// TIA Portal project "项目1" (V14)

(* hardware
DEVICE "S7-1200 station_1"  S7-1200 Station
   slot 0: "Rack_0"  S7-1200 Rack  Rack  V1.0
   slot 1: "PLC_xingneng"  CPU 1214C DC/DC/DC  6ES7 214-1AG40-0XB0  V4.2
   slot 2: "DI 16/DQ 16x24VDC_1"  6ES7 223-1BL32-0XB0  V2.0
   slot 3: "DI 16/DQ 16x24VDC_2"  6ES7 223-1BL32-0XB0  V2.0
   slot 4: "AI 4x13BIT/AQ 2x14BIT_1"  6ES7 234-4HE32-0XB0  V2.0
   slot 5: "AI 4x13BIT/AQ 2x14BIT_2"  6ES7 234-4HE32-0XB0  V2.0
DEVICE "v90-pn-1"  GSD.Device.PN
   slot 0: "SINAMICS-V90-PN"  SINAMICS V90 PN V1.0  6SL3 210-5Fxxx-xxFx  V1.00
      slot 0: "SINAMICS V90 PN V1.0"  SINAMICS V90 PN V1.0
      slot 1: "驱动_1"  Drive
         slot 0: "模块访问点"  Module Access Point
         slot 1: "没有 PROFIsafe"  without PROFIsafe
      slot 1: "PN-IO"  PN-IO
         slot 1: "端口1"  Port 1
         slot 2: "端口2"  Port 2
   slot 0: "机架"  Rack  V1.0
   slot 2: "标准报文3, PZD-5/9"  Standard telegram 3, PZD-5/9
*)

// ===== PLC "PLC_xingneng"  CPU 1214C DC/DC/DC =====
// protected blocks, not shown: "buffer"

VAR_GLOBAL   // PLC tag table "默认变量表"
   "输入轴扭矩传感器" AT %IW128 : Int;
   "输出轴扭矩传感器Min_A" AT %IW130 : Int;
   "轴_1_LowHwLimitSwitch" AT %I0.3 : Bool;
   "轴_1_HighHwLimitSwitch" AT %I0.4 : Bool;
   "轴_1_参考点开关" AT %I0.2 : Bool;
   "轴_2_LowHwLimitSwitch" AT %I0.6 : Bool;
   "轴_2_HighHwLimitSwitch" AT %I0.7 : Bool;
   "轴_2_参考点开关" AT %I0.5 : Bool;
   "输出轴扭矩传感器Max_B" AT %IW132 : Int;
   "电流计" AT %IW134 : Int;
   "Tag_45" AT %I11.0 : Bool;
   "Tag_46" AT %I11.3 : Bool;
   "输入轴角度" AT %ID1000 : DInt;
   "Tag_70" AT %ID100 : DInt;
   "Tag_80" AT %ID0 : DWord;
   "Tag_86" AT %IW0 : Word;
   "Tag_87" AT %IW8 : Word;
   "Tag_88" AT %IW12 : Word;
   "工件在位" AT %I3.6 : Bool;
   "输入移报警" AT %I2.0 : Bool;
   "高度适配轴参考点" AT %I2.1 : Bool;
   "输出移报警" AT %I2.2 : Bool;
   "高度适配轴上限" AT %I2.3 : Bool;
   "输入旋报警" AT %I2.4 : Bool;
   "高度适配轴下限" AT %I2.5 : Bool;
   "输出旋报警" AT %I2.6 : Bool;
   "输出旋到位" AT %I2.7 : Bool;
   "抱花键进到位" AT %I3.0 : Bool;
   "抱花键退到位" AT %I3.1 : Bool;
   "摆臂1进到位" AT %I3.2 : Bool;
   "摆臂1退到位" AT %I3.3 : Bool;
   "摆臂2进到位" AT %I3.4 : Bool;
   "摆臂2退到位" AT %I3.5 : Bool;
   "振动进到位" AT %I4.0 : Bool;
   "振动退到位" AT %I4.1 : Bool;
   "升降门进到位" AT %I4.2 : Bool;
   "升降门退到位" AT %I4.3 : Bool;
   "急停" AT %I5.0 : Bool;
   "启动" AT %I5.1 : Bool;
   "复位" AT %I5.3 : Bool;
   "输出轴角度" AT %ID1004 : DInt;
   "Tag_1" AT %IW138 : Int;
   "ECU传感器" AT %IW136 : Int;
   "安全光栅" AT %I3.7 : Bool;
   "轴_5_Drive_IN" AT %I68.0 : "PD_TEL3_IN";
   "高度适配轴错误" AT %I1.5 : Bool;
   "产品定位缸进位" AT %I4.4 : Bool;
   "产品定位缸退位" AT %I4.5 : Bool;
   "右震动检测进位" AT %I4.6 : Bool;
   "右震动检测退位" AT %I4.7 : Bool;
   "Tag_116" AT %I5.4 : Bool;
   "工件在位检测" AT %I5.5 : Bool;
   "轴_1_Pulse_Up" AT %Q0.0 : Bool;
   "轴_1_Pulse_Down" AT %Q0.1 : Bool;
   "轴_2_脉冲" AT %Q0.2 : Bool;
   "轴_2_方向" AT %Q0.3 : Bool;
   "Tag_25" AT %QW128 : Word;
   "Tag_26" AT %QW130 : Int;
   "Tag_27" AT %QW80 : Int;
   "Tag_53" AT %Q6.0 : Bool;
   "Tag_54" AT %Q6.1 : Bool;
   "Tag_55" AT %Q6.2 : Bool;
   "Tag_56" AT %Q6.3 : Bool;
   "Tag_57" AT %Q6.4 : Bool;
   "Tag_58" AT %Q6.5 : Bool;
   "Tag_59" AT %Q6.6 : Bool;
   "Tag_60" AT %Q6.7 : Bool;
   "Tag_79" AT %QD0 : DWord;
   "Tag_82" AT %QW0 : Word;
   "Tag_83" AT %QW8 : Word;
   "Tag_84" AT %QW12 : Word;
   "Tag_85" AT %QW2 : Word;
   "控制器转速" AT %Q0.6 : Bool;
   "carPulse" AT %Q0.4 : Bool;
   "控制器切换" AT %Q1.0 : Bool;
   "输入移警清" AT %Q2.0 : Bool;
   "输出移警清" AT %Q2.1 : Bool;
   "输入旋模式" AT %Q2.3 : Bool;
   "输入旋警清" AT %Q2.4 : Bool;
   "输出旋模式" AT %Q2.6 : Bool;
   "输出旋警清" AT %Q2.7 : Bool;
   "抱花键" AT %Q4.0 : Bool;
   "摆臂进" AT %Q4.1 : Bool;
   "摆臂退" AT %Q4.2 : Bool;
   "振动" AT %Q4.5 : Bool;
   "升降门进" AT %Q4.3 : Bool;
   "升降门退" AT %Q4.4 : Bool;
   "黄" AT %Q3.0 : Bool;
   "绿" AT %Q3.1 : Bool;
   "红" AT %Q3.2 : Bool;
   "蜂鸣" AT %Q3.3 : Bool;
   "输入旋速" AT %Q2.2 : Bool;
   "输出旋速" AT %Q2.5 : Bool;
   "PowerECU" AT %Q0.5 : Bool;
   "switch" AT %Q3.5 : Bool;
   "0-1KHZ占空比" AT %QW132 : Int;
   "30V电源" AT %QW134 : Int;
   "Tag_7" AT %QD4 : DWord;
   "resetAxis1" AT %Q1.6 : Bool;
   "resetAxis2" AT %Q1.7 : Bool;
   "轴_4_方向" AT %Q0.7 : Bool;
   "轴_5_Drive_OUT" AT %Q64.0 : "PD_TEL3_OUT";
   "产品高度适配轴JOG+" AT %Q7.0 : Bool;
   "产品高度适配轴故障复位" AT %Q5.4 : Bool;
   "高度适配轴JOG+" AT %Q5.6 : Bool;
   "高度适配轴JOG-" AT %Q5.7 : Bool;
   "高度适配轴回原点" AT %Q5.5 : Bool;
   "产品定位缸进" AT %Q5.0 : Bool;
   "产品定位缸退" AT %Q5.1 : Bool;
   "右震动检测缸进" AT %Q5.2 : Bool;
   "右震动检测缸退" AT %Q5.3 : Bool;
   "电机方向" AT %Q4.6 : Bool;
   "电机控制" AT %Q4.7 : Bool;
   "funtionStatus" AT %MB10 : SInt;
   "Tag_18" AT %M0.0 : Bool;
   "Tag_19" AT %M0.1 : Bool;
   "Tag_20" AT %M0.2 : Bool;
   "Tag_21" AT %M0.3 : Bool;
   "Tag_22" AT %M0.7 : Bool;
   "Tag_23" AT %M0.6 : Bool;
   "Tag_24" AT %M0.4 : Bool;
   "Tag_30" AT %M0.5 : Bool;
   "torqueInput" AT %MD100 : Real;
   "torqueOutputA" AT %MD104 : Real;
   "Tag_33" AT %MD200 : Real;
   "Tag_34" AT %MD204 : Real;
   "Tag_35" AT %MD206 : Real;
   "Tag_36" AT %MD106 : Real;
   "torqueOutputB" AT %MD108 : Real;
   "current" AT %MD112 : Real;
   "Tag_3" AT %M10.0 : Bool;
   "Tag_42" AT %M11.0 : Bool;
   "Tag_43" AT %M12.0 : Bool;
   "Tag_44" AT %M10.1 : Bool;
   "Tag_47" AT %M10.2 : Bool;
   "Tag_48" AT %M10.3 : Bool;
   "Tag_51" AT %MW20 : Word;
   "Tag_62" AT %M10.4 : Bool;
   "Tag_64" AT %M10.5 : Bool;
   "Tag_65" AT %M12.3 : Bool;
   "Tag_66" AT %M13.0 : Bool;
   "Tag_67" AT %M11.1 : Bool;
   "Tag_68" AT %M10.6 : Bool;
   "Tag_69" AT %MW30 : Word;
   "Tag_71" AT %M30.0 : Bool;
   "Tag_72" AT %M35.0 : Bool;
   "Tag_73" AT %M30.5 : Bool;
   "Tag_74" AT %M35.6 : Bool;
   "Tag_75" AT %M35.5 : Bool;
   "Tag_76" AT %MW36 : Word;
   "Tag_77" AT %MW40 : Word;
   "Tag_89" AT %MW32 : Word;
   "Tag_28" AT %M30.7 : Bool;
   "Tag_29" AT %M1.0 : Bool;
   "Tag_49" AT %M1.1 : Bool;
   "Tag_50" AT %M1.2 : Bool;
   "Tag_61" AT %M1.3 : Bool;
   "Tag_90" AT %MB1 : Byte;
   "Tag_16" AT %M2.0 : Bool;
   "Tag_17" AT %M1.4 : Bool;
   "Tag_41" AT %M1.7 : Bool;
   "angleInput" AT %MD150 : Real;
   "angleOutput" AT %MD154 : Real;
   "sensorA" AT %MD116 : Real;
   "sensorB" AT %MD120 : Real;
   "carSpeed" AT %MD1000 : Real;
   "Tag_8" AT %M11.2 : Bool;
   "Tag_9" AT %M11.3 : Bool;
   "Tag_10" AT %M11.4 : Bool;
   "Tag_11" AT %M11.5 : Bool;
   "Tag_12" AT %M11.6 : Bool;
   "Tag_13" AT %M11.7 : Bool;
   "Tag_31" AT %M12.1 : Bool;
   "Tag_32" AT %M13.1 : Bool;
   "Tag_37" AT %M13.2 : Bool;
   "Tag_38" AT %M13.3 : Bool;
   "Tag_52" AT %M13.4 : Bool;
   "Tag_78" AT %M13.5 : Bool;
   "Tag_81" AT %M13.6 : Bool;
   "Tag_91" AT %M13.7 : Bool;
   "Tag_92" AT %MB11 : Byte;
   "Tag_93" AT %MB12 : Byte;
   "Tag_94" AT %MB13 : Byte;
   "Tag_95" AT %M2.1 : Bool;
   "carSpeed(1)" AT %MD5 : Real;
   "Tag_97" AT %M2.2 : Bool;
   "光栅故障" AT %M3.0 : Bool;
   "Tag_96" AT %M12.2 : Bool;
   "Tag_98" AT %MW1004 : Word;
   "Tag_99" AT %M300.0 : Bool;
   "Tag_100" AT %MW11 : Word;
   "Tag_101" AT %MD11 : DWord;
   "Tag_102" AT %M2.3 : Bool;
   "Tag_104" AT %M14.0 : Bool;
   "Tag_108" AT %M14.1 : Bool;
   "Tag_113" AT %M14.2 : Bool;
   "Tag_114" AT %M14.3 : Bool;
   "Tag_115" AT %M14.4 : Bool;
   "Tag_117" AT %M2.4 : Bool;
   "Tag_118" AT %M2.5 : Bool;
   "Tag_119" AT %M300.1 : Bool;
   "Tag_120" AT %M310.0 : Bool;
   "Tag_103" AT %M310.1 : Bool;
   "Tag_105" AT %M310.3 : Bool;
   "轴_5当前位移" AT %MD2000 : Real;
   "Tag_106" AT %M14.5 : Bool;
   "轴_1当前位移" AT %MD2004 : DWord;
   "轴_2当前位移" AT %MD2008 : DWord;
   "Tag_4" AT %M2012.0 : Bool;
   "Tag_5" AT %MD1004 : Real;
   "Tag_6" AT %MW2000 : Word;
   "Tag_107" AT %MW3000 : Word;
   "Tag_109" AT %MD2500 : DInt;
   "Tag_110" AT %MB2503 : Byte;
   "Tag_111" AT %M200.0 : Bool;
   "Tag_112" AT %M200.1 : Bool;
   "Tag_121" AT %M200.2 : Bool;
   "Tag_122" AT %M200.3 : Bool;
END_VAR

TYPE "In_config"
VERSION : 0.1
   STRUCT
      inAxis_接近位移 : Real;
      inAxis_接近速度 : Real;
      inAxis_套入位移 : Real;
      inAxis_套入速度 : Real;
      outAxis_接近位置 : Real;
      outAxis_接近速度 : Real;
      outAxis_套入位置 : Real;
      outAxis_套入速度 : Real;
   END_STRUCT;
END_TYPE

TYPE "In_swing_config"
VERSION : 0.1
   STRUCT
      启用状态 : Real;
      摆动速度 : Real;
      摆动角度 : Real;
      保护扭矩 : Real;
   END_STRUCT;
END_TYPE

TYPE "Fixture_transfer_config"
VERSION : 0.1
   STRUCT
      定位位置 : Real;
      定位速度 : Real;
   END_STRUCT;
END_TYPE

TYPE "Test_No_Load_CFG"
VERSION : 0.1
   STRUCT
      启用助力 : Real := 0.0;
      空载速度 : Real := 0.0;
      空载位移 : Real := 0.0;
      扭矩保护 : Real := 0.0;
   END_STRUCT;
END_TYPE

TYPE "Test_Function_CFG"
VERSION : 0.1
   STRUCT
      试验速度 : Real;
      试验角度 : Real;
      负载扭矩 : Real;
      保护扭矩 : Real;
   END_STRUCT;
END_TYPE

TYPE "Test_Input&Output_Characteristics_CFG"
VERSION : 0.1
   STRUCT
      试验速度 : Real;
      换向扭矩 : Real;
      模拟车速 : Real;
      模拟转速 : Real;
   END_STRUCT;
END_TYPE

TYPE "Test_NVH"
VERSION : 0.1
   STRUCT
      检测点1 : Real;
      检测点2 : Real;
      正向检测时间 : Real;
      逆向检测时间 : Real;
   END_STRUCT;
END_TYPE

DATA_BLOCK "auto_4_DB_1"   // DB1
{ S7_Optimized_Access := 'TRUE' }
VERSION : 0.1
// stored: InstanceOfName 逆向空载
"逆向空载"
BEGIN
END_DATA_BLOCK

DATA_BLOCK "Data_sendset"   // DB2
{ S7_Optimized_Access := 'TRUE' }
VERSION : 0.1
   VAR
      REQ : Bool;
      CONT : Bool := 1;
      LEN : UInt := 8;
      DONE : Bool;
      BUSY : Bool;
      ERROR : Bool;
      STATUS : Word;
      COM_RST : Bool;
      CONNECT : TCON_Param;
      NUM : DInt;
      X : Real;
      Y : Real;
      Z : Real;
   END_VAR
BEGIN
END_DATA_BLOCK

DATA_BLOCK "Data_send_0"   // DB3
{ S7_Optimized_Access := 'FALSE' }
VERSION : 0.1
   VAR
      ai : Array[0..99] of Real;
   END_VAR
BEGIN
END_DATA_BLOCK

DATA_BLOCK "auto_6_DB"   // DB4
{ S7_Optimized_Access := 'TRUE' }
VERSION : 0.1
// stored: InstanceOfName 固定工件
"固定工件"
BEGIN
END_DATA_BLOCK

DATA_BLOCK "Data_send_1"   // DB5
{ S7_Optimized_Access := 'FALSE' }
VERSION : 0.1
   VAR
      ai : Array[0..99] of Real;
   END_VAR
BEGIN
END_DATA_BLOCK

DATA_BLOCK "reset_DB"   // DB6
{ S7_Optimized_Access := 'TRUE' }
VERSION : 0.1
// stored: InstanceOfName reset
"reset"
BEGIN
END_DATA_BLOCK

DATA_BLOCK "MD_data"   // DB7
{ S7_Optimized_Access := 'FALSE' }
VERSION : 0.1
   VAR
      输入扭矩传感器参数 : Array[0..1] of Real;
      输出扭矩传感器参数A : Array[0..1] of Real;
      输出扭矩传感器参数B : Array[0..1] of Real;
      电流传感器参数 : Array[0..1] of Real;
      轴自动参数 : "In_config";
      输入轴移栽手动速度 : Array[0..3] of Real;
      输入轴旋转参数 : Array[0..3] of Real;
      工装定位参数 : "Fixture_transfer_config";
      工装手动参数 : Array[0..3] of Real;
      空载试验参数 : "Test_No_Load_CFG";
      功能试验参数 : "Test_Function_CFG";
      力特性试验参数 : "Test_Input&Output_Characteristics_CFG";
      逆向空载试验参数 : "Test_No_Load_CFG";
      振动NVH试验参数 : "Test_NVH";
      辅助参数 : Array[0..3] of Real;
   END_VAR
BEGIN
   输入扭矩传感器参数[1] := 18.8;   // 校验值19.2
   输出扭矩传感器参数A[1] := 10.0;   // 校验值9.5
   输出扭矩传感器参数B[1] := 113.0;   // 校验值97.0
   电流传感器参数[0] := -100.0;
   电流传感器参数[1] := 100.0;
   // 辅助参数[0] : 安全门开启
END_DATA_BLOCK

DATA_BLOCK "Data_recset"   // DB8
{ S7_Optimized_Access := 'TRUE' }
VERSION : 0.1
   VAR
      REQ : Bool;
      CONT : Bool := 1;
      LEN : UInt := 8;
      DONE : Bool;
      BUSY : Bool;
      ERROR : Bool;
      STATUS : Word;
      COM_RST : Bool;
      CONNECT : TCON_Param;
      NUM : UDInt;
      X : Real;
      Y : Real;
      Z : Real;
   END_VAR
BEGIN
END_DATA_BLOCK

DATA_BLOCK "alarm_DB"   // DB10
{ S7_Optimized_Access := 'TRUE' }
VERSION : 0.1
// stored: InstanceOfName alarm
"alarm"
BEGIN
END_DATA_BLOCK

DATA_BLOCK "auto_7_DB"   // DB12
{ S7_Optimized_Access := 'TRUE' }
VERSION : 0.1
// stored: InstanceOfName 振动检测
"振动检测"
BEGIN
END_DATA_BLOCK

DATA_BLOCK "Data_set"   // DB21
{ S7_Optimized_Access := 'TRUE' }
VERSION : 0.1
   VAR
      "real" : Array[0..16] of Real;
   END_VAR
BEGIN
   "real"[0] := 2.0;
END_DATA_BLOCK

DATA_BLOCK "manual_DB"   // DB22
{ S7_Optimized_Access := 'TRUE' }
VERSION : 0.1
// stored: InstanceOfName manual
"manual"
BEGIN
END_DATA_BLOCK

DATA_BLOCK "auto_8_DB"   // DB23
{ S7_Optimized_Access := 'TRUE' }
VERSION : 0.1
// stored: InstanceOfName 功能
"功能"
BEGIN
END_DATA_BLOCK

DATA_BLOCK "auto_1_DB"   // DB28
{ S7_Optimized_Access := 'TRUE' }
VERSION : 0.1
// stored: InstanceOfName 套输入轴花键
"套输入轴花键"
BEGIN
END_DATA_BLOCK

DATA_BLOCK "auto_2_DB"   // DB31
{ S7_Optimized_Access := 'TRUE' }
VERSION : 0.1
// stored: InstanceOfName 套输出轴花键
"套输出轴花键"
BEGIN
END_DATA_BLOCK

DATA_BLOCK "motor_run_DB"   // DB32
{ S7_Optimized_Access := 'TRUE' }
VERSION : 0.1
// stored: InstanceOfName motor_m
"motor_m"
BEGIN
END_DATA_BLOCK

DATA_BLOCK "motor_run_DB_1"   // DB33
{ S7_Optimized_Access := 'TRUE' }
VERSION : 0.1
// stored: InstanceOfName motor_m
"motor_m"
BEGIN
END_DATA_BLOCK

DATA_BLOCK "motor_run_DB_2"   // DB34
{ S7_Optimized_Access := 'TRUE' }
VERSION : 0.1
// stored: InstanceOfName motor_m
"motor_m"
BEGIN
END_DATA_BLOCK

DATA_BLOCK "motor_m_DB"   // DB35
{ S7_Optimized_Access := 'TRUE' }
VERSION : 0.1
// stored: InstanceOfName motor_m
"motor_m"
BEGIN
END_DATA_BLOCK

DATA_BLOCK "auto_3_DB"   // DB37
{ S7_Optimized_Access := 'TRUE' }
VERSION : 0.1
// stored: InstanceOfName 空载与标定
"空载与标定"
BEGIN
END_DATA_BLOCK

DATA_BLOCK "auto_4_DB"   // DB39
{ S7_Optimized_Access := 'TRUE' }
VERSION : 0.1
// stored: InstanceOfName 力特性
"力特性"
BEGIN
END_DATA_BLOCK

DATA_BLOCK "auto_100_DB"   // DB45
{ S7_Optimized_Access := 'TRUE' }
VERSION : 0.1
// stored: InstanceOfName auto_100
"auto_100"
BEGIN
END_DATA_BLOCK

DATA_BLOCK "找零_DB"   // DB66
{ S7_Optimized_Access := 'TRUE' }
VERSION : 0.1
// stored: InstanceOfName 找零
"找零"
BEGIN
END_DATA_BLOCK

DATA_BLOCK "MD_data_Rapid"   // DB70
{ S7_Optimized_Access := 'FALSE' }
VERSION : 0.1
   VAR
      设备编号 : Int;
      产品型号 : Int;
      设备状态 : Int;
      错误代码 : Int;
      当前曲线 : Int;
      传感器标定值 : Array[0..11] of Real;
   END_VAR
BEGIN
   // 传感器标定值[0] : 输入轴驱动伺服位移
   // 传感器标定值[1] : 输入轴移载伺服位移
   // 传感器标定值[2] : 工装移载伺服位移
   // 传感器标定值[3] : 输入轴旋转角度
   // 传感器标定值[4] : 输入轴扭矩
   // 传感器标定值[5] : 输出轴扭矩小量程
   // 传感器标定值[6] : 输出轴扭矩大量程
   // 传感器标定值[7] : 吸收电流
   // 传感器标定值[8] : factorSensorT1
   // 传感器标定值[9] : 输出轴旋转角度
   // 传感器标定值[10] : 输出轴移栽位移
   // 传感器标定值[11] : factorSensorT2
END_DATA_BLOCK

DATA_BLOCK "buffer_dataSet"   // DB100
{ S7_Optimized_Access := 'FALSE' }
VERSION : 0.1
   VAR
      factorInputTorque : Real := 20.0;
      factorOutputTorqueA : Real := 10.0;
      factorOutputTorqueB : Real := 100.0;
      factorCurrent : Real := 100.0;
      factorSensor : Real := 20.0;
      offsetInputTorqueRight : Real;
      offsetInputTorqueLeft : Real;
      offsetOutputTorqueRightA : Real;
      offsetOutputTorqueLeftA : Real;
      offsetOutputTorqueRightB : Real;
      offsetOutputTorqueLeftB : Real;
      offsetCurrent : Real;
      offsetSensor : Real;
      set_7 : Real;
      set_8 : Real;
      set_9 : Real;
      set_10 : Real;
      set_11 : Real;
      set_12 : Real;
      set_13 : Real;
      distanceInputNear : Real;
      distanceOutputNear : Real;
      distanceInputPoint : Real;
      distanceOutputPoint : Real;
      door : Real;
      voltageECU : Real;
      funtionSpeed : Real;
      funtionAngle : Real;
      funtionSpeedCar : Real;
      funtionLoad : Real;
      forceTorque : Real;
      noloadSpeed : Real;
      noloadAngle : Real;
      noloadPowerECU : Real;
      reverseloadSpeed : Real;
      reverseloadAngle : Real;
      reverseloadPowerECU : Real;
   END_VAR
BEGIN
END_DATA_BLOCK

DATA_BLOCK "buffer_dataSend"   // DB101
{ S7_Optimized_Access := 'FALSE' }
VERSION : 0.1
   VAR
      dataSend : Array[0..51] of Real;
   END_VAR
BEGIN
END_DATA_BLOCK

// folder: System blocks/Program resources

DATA_BLOCK "IEC_Timer_0_DB_1"   // DB51
{ S7_Optimized_Access := 'TRUE' }
AUTHOR : Simatic
FAMILY : IEC
NAME : IEC_TMR
VERSION : 1.0
// stored: InstanceOfName IEC_TIMER
"IEC_TIMER"
BEGIN
END_DATA_BLOCK

DATA_BLOCK "IEC_Timer_0_DB_3"   // DB59
{ S7_Optimized_Access := 'TRUE' }
AUTHOR : Simatic
FAMILY : IEC
NAME : IEC_TMR
VERSION : 1.0
// stored: InstanceOfName IEC_TIMER
"IEC_TIMER"
BEGIN
END_DATA_BLOCK

DATA_BLOCK "IEC_Timer_0_DB_4"   // DB63
{ S7_Optimized_Access := 'TRUE' }
AUTHOR : Simatic
FAMILY : IEC
NAME : IEC_TMR
VERSION : 1.0
// stored: InstanceOfName IEC_TIMER
"IEC_TIMER"
BEGIN
END_DATA_BLOCK

DATA_BLOCK "IEC_Timer_0_DB_2"   // DB64
{ S7_Optimized_Access := 'TRUE' }
AUTHOR : Simatic
FAMILY : IEC
NAME : IEC_TMR
VERSION : 1.0
// stored: InstanceOfName IEC_TIMER
"IEC_TIMER"
BEGIN
END_DATA_BLOCK

DATA_BLOCK "IEC_Timer_0_DB_5"   // DB65
{ S7_Optimized_Access := 'TRUE' }
AUTHOR : Simatic
FAMILY : IEC
NAME : IEC_TMR
VERSION : 1.0
// stored: InstanceOfName IEC_TIMER
"IEC_TIMER"
BEGIN
END_DATA_BLOCK

// folder: (top level)

DATA_BLOCK "轴_1"   // DB14, Motion_DB
{ S7_Optimized_Access := 'TRUE' }
AUTHOR : SIMATIC
FAMILY : BasicMC
NAME : TO_PosAx
VERSION : 6.0
// stored: InstanceOfName TO_PositioningAxis
"TO_PositioningAxis"
BEGIN
   // Axis.DirectionOutputEnabledCU = TRUE
   // Axis.OnlinePtoModeCUEnumValue = PTO（脉冲 A 和方向 B）
   // Axis.OnlinePtoModeCU = 16#0000_0002
   // Axis.SelectPTO = 0
   // Axis.LeadScrew = 5.0
   // Axis.LeadScrew.Distance = 1013
   // Axis.PositionLimitsMinPosition = -10000.0
   // Axis.PositionLimitsMinPosition.Distance = 1013
   // Axis.PositionLimitsMaxPosition = 10000.0
   // Axis.PositionLimitsMaxPosition.Distance = 1013
   // Axis.HomingOffset = 0.0
   // Axis.HomingOffset.Distance = 1013
   // Axis.HomingFastVelocity = 30.0
   // Axis.HomingFastVelocity.Distance = 1013
   // Axis.NormalizedMaxVelocity = 50.0
   // Axis.NormalizedMaxVelocity.Distance = 1013
   // Axis.NormalizedMaxVelocity.Time = 0
   // Axis.MaxVelocityReadOnly = 50.0
   // Axis.MaxVelocityReadOnly.Distance = 1013
   // Axis.NormalizedMinVelocity = 1.0
   // Axis.NormalizedMinVelocity.Distance = 1013
   // Axis.NormalizedMinVelocity.Time = 0
   // Axis.MinVelocityReadOnly = 1.0
   // Axis.MinVelocityReadOnly.Distance = 1013
   // Axis.Acceleration = 245.0
   // Axis.Acceleration.Distance = 1013
   // Axis.RampUpTime = 0.2
   // Axis.Deceleration = 245.0
   // Axis.Deceleration.Distance = 1013
   // Axis.RampDownTime = 0.2
   // Axis.RoundUpTime = 0.0
   // Axis.Jerk = 0.0
   // Axis.Jerk.Distance = 1013
   // Axis.RampDownTimeEmergency = 0.1
   // Axis.DecelerationEmergency = 490.0
   // Axis.DecelerationEmergency.Distance = 1013
   // Axis.HomingSlowVelocity = 10.0
   // Axis.HomingSlowVelocity.Distance = 1013
   // Axis.LengthUnitNormalized.Distance = 1013
   // Axis.LengthUnitNormalized.Time = 0
   // Pulse.OutputSourceCU = 16#0000_0000
   // Pulse.MaxFrequencyCU = 100000.0
   // Pulse.MinFrequencyCU = 1.0
   // Pulse.MaxDeltaFrequencyCU = 9.5E+9
   // Pulse.MinDeltaFrequencyCU = 0.005
   // Pulse.MaxDeltaDeltaFrequencyCU = 1.0E+10
   // Pulse.MinDeltaDeltaFrequencyCU = 0.004
   // Axis.SelectedChannel1EnumCU = %Q0.0
   // Axis.SelectedChannel2EnumCU = %Q0.1
   // Axis.PositionLimitsMin_AddressCU = %I0.3
   // Axis.PositionLimitsMax_AddressCU = %I0.4
   // Axis.PassiveHomingReferencePointSwitch_AddressCU = %I0.2
   // Axis.HomingReferencePointSwitch_AddressCU = %I0.2
END_DATA_BLOCK

DATA_BLOCK "轴_2"   // DB15, Motion_DB
{ S7_Optimized_Access := 'TRUE' }
AUTHOR : SIMATIC
FAMILY : BasicMC
NAME : TO_PosAx
VERSION : 6.0
// stored: InstanceOfName TO_PositioningAxis
"TO_PositioningAxis"
BEGIN
   // Axis.DirectionOutputEnabledCU = TRUE
   // Axis.OnlinePtoModeCUEnumValue = PTO（脉冲 A 和方向 B）
   // Axis.OnlinePtoModeCU = 16#0000_0002
   // Axis.SelectPTO = 1
   // Axis.LeadScrew = 5.0
   // Axis.LeadScrew.Distance = 1013
   // Axis.PositionLimitsMinPosition = -10000.0
   // Axis.PositionLimitsMinPosition.Distance = 1013
   // Axis.PositionLimitsMaxPosition = 10000.0
   // Axis.PositionLimitsMaxPosition.Distance = 1013
   // Axis.HomingOffset = 0.0
   // Axis.HomingOffset.Distance = 1013
   // Axis.HomingFastVelocity = 20.0
   // Axis.HomingFastVelocity.Distance = 1013
   // Axis.NormalizedMaxVelocity = 50.0
   // Axis.NormalizedMaxVelocity.Distance = 1013
   // Axis.NormalizedMaxVelocity.Time = 0
   // Axis.MaxVelocityReadOnly = 50.0
   // Axis.MaxVelocityReadOnly.Distance = 1013
   // Axis.NormalizedMinVelocity = 1.0
   // Axis.NormalizedMinVelocity.Distance = 1013
   // Axis.NormalizedMinVelocity.Time = 0
   // Axis.MinVelocityReadOnly = 1.0
   // Axis.MinVelocityReadOnly.Distance = 1013
   // Axis.Acceleration = 245.0
   // Axis.Acceleration.Distance = 1013
   // Axis.RampUpTime = 0.2
   // Axis.Deceleration = 245.0
   // Axis.Deceleration.Distance = 1013
   // Axis.RampDownTime = 0.2
   // Axis.RoundUpTime = 0.0
   // Axis.Jerk = 0.0
   // Axis.Jerk.Distance = 1013
   // Axis.RampDownTimeEmergency = 0.1
   // Axis.DecelerationEmergency = 490.0
   // Axis.DecelerationEmergency.Distance = 1013
   // Axis.HomingSlowVelocity = 10.0
   // Axis.HomingSlowVelocity.Distance = 1013
   // Axis.LengthUnitNormalized.Distance = 1013
   // Axis.LengthUnitNormalized.Time = 0
   // Pulse.OutputSourceCU = 16#0000_0000
   // Pulse.MaxFrequencyCU = 100000.0
   // Pulse.MinFrequencyCU = 1.0
   // Pulse.MaxDeltaFrequencyCU = 9.5E+9
   // Pulse.MinDeltaFrequencyCU = 0.005
   // Pulse.MaxDeltaDeltaFrequencyCU = 1.0E+10
   // Pulse.MinDeltaDeltaFrequencyCU = 0.004
   // Axis.OnlinePtoIndexCU = 1
   // Axis.SelectedChannel1EnumCU = %Q0.2
   // Axis.SelectedChannel2EnumCU = %Q0.3
   // Axis.PositionLimitsMin_AddressCU = %I0.6
   // Axis.PositionLimitsMax_AddressCU = %I0.7
   // Axis.PassiveHomingReferencePointSwitch_AddressCU = %I0.5
   // Axis.HomingReferencePointSwitch_AddressCU = %I0.5
END_DATA_BLOCK

DATA_BLOCK "轴_3"   // DB46, Motion_DB
{ S7_Optimized_Access := 'TRUE' }
AUTHOR : SIMATIC
FAMILY : BasicMC
NAME : TO_PosAx
VERSION : 6.0
// stored: InstanceOfName TO_PositioningAxis
"TO_PositioningAxis"
BEGIN
   // Axis.SelectedChannel2EnumCU = %Q0.3
   // Axis.OnlinePtoModeCUEnumValue = PTO（脉冲 A 和方向 B）
   // Axis.OnlinePtoModeCU = 16#0000_0002
   // Axis.SelectPTO = 2
   // Axis.LengthUnit.LastDistance = -1
   // Axis.LeadScrew = 10.0
   // Axis.LeadScrew.Distance = -1
   // Axis.PositionLimitsMinPosition = -1.0E+6
   // Axis.PositionLimitsMinPosition.Distance = -1
   // Axis.PositionLimitsMaxPosition = 1.0E+6
   // Axis.PositionLimitsMaxPosition.Distance = -1
   // Axis.HomingOffset = 0.0
   // Axis.HomingOffset.Distance = -1
   // Axis.HomingFastVelocity = 20000.0
   // Axis.HomingFastVelocity.Distance = -1
   // Axis.NormalizedMaxVelocity = 500.0
   // Axis.NormalizedMaxVelocity.Distance = -1
   // Axis.NormalizedMaxVelocity.Time = 0
   // Axis.MaxVelocityReadOnly = 500.0
   // Axis.MaxVelocityReadOnly.Distance = -1
   // Axis.NormalizedMinVelocity = 1.0
   // Axis.NormalizedMinVelocity.Distance = -1
   // Axis.NormalizedMinVelocity.Time = 0
   // Axis.MinVelocityReadOnly = 1.0
   // Axis.MinVelocityReadOnly.Distance = -1
   // Axis.Acceleration = 4990.0
   // Axis.Acceleration.Distance = -1
   // Axis.RampUpTime = 0.1
   // Axis.Deceleration = 4990.0
   // Axis.Deceleration.Distance = -1
   // Axis.RampDownTime = 0.1
   // Axis.RoundUpTime = 0.0
   // Axis.Jerk = 0.0
   // Axis.Jerk.Distance = -1
   // Axis.RampDownTimeEmergency = 0.1
   // Axis.DecelerationEmergency = 4990.0
   // Axis.DecelerationEmergency.Distance = -1
   // Axis.HomingSlowVelocity = 4000.0
   // Axis.HomingSlowVelocity.Distance = -1
   // Axis.LengthUnitNormalized.Distance = -1
   // Axis.LengthUnitNormalized.Time = 0
   // Pulse.OutputSourceCU = 16#0000_0000
   // Pulse.MaxFrequencyCU = 30000.0
   // Pulse.MinFrequencyCU = 1.0
   // Pulse.MaxDeltaFrequencyCU = 9.5E+9
   // Pulse.MinDeltaFrequencyCU = 0.005
   // Pulse.MaxDeltaDeltaFrequencyCU = 1.0E+10
   // Pulse.MinDeltaDeltaFrequencyCU = 0.004
   // Axis.OnlinePtoIndexCU = 2
   // Axis.SelectedChannel1EnumCU = %Q0.4
END_DATA_BLOCK

DATA_BLOCK "轴_5"   // DB52, Motion_DB
{ S7_Optimized_Access := 'TRUE' }
AUTHOR : SIMATIC
FAMILY : BasicMC
NAME : TO_PosAx
VERSION : 6.0
// stored: InstanceOfName TO_PositioningAxis
"TO_PositioningAxis"
BEGIN
   // Axis.PositionLimitsMax_AddressCU = %I2.3
   // Axis.PositionLimitsMin_AddressCU = %I2.5
   // Axis.HomingReferencePointSwitch_AddressCU = %I2.1
   // Axis.Encoder.TelegramAddressOutCU = %Q64.0
   // Axis.Encoder.TelegramAddressInCU = %I68.0
   // Axis.Encoder.OutputAddress = 64
   // Axis.Encoder.InputAddress = 68
   // Axis.Encoder.DoNameCU = SINAMICS-V90-PN.驱动_1
   // Axis.Drive.OutputAddress = 64
   // Axis.Drive.InputAddress = 68
   // Axis.Drive.TelegramAddressOutCU = %Q64.0
   // Axis.Drive.TelegramAddressInCU = %I68.0
   // Axis.Drive.TelegramType = 2
   // Axis.Drive.DoNameCU = SINAMICS-V90-PN.驱动_1
   // Axis.LengthUnitNormalized.Distance = 1013
   // Axis.Encoder.SelectedHscIndexCU = -1
   // Axis.Encoder.DbTypeCU = Classic
   // Axis.Drive.DbTypeCU = Classic
END_DATA_BLOCK

DATA_BLOCK "轴_4"   // DB53, Motion_DB
{ S7_Optimized_Access := 'TRUE' }
AUTHOR : SIMATIC
FAMILY : BasicMC
NAME : TO_PosAx
VERSION : 6.0
// stored: InstanceOfName TO_PositioningAxis
"TO_PositioningAxis"
BEGIN
   // Axis.SelectedChannel2EnumCU = %Q0.7
   // Axis.LengthUnit.LastDistance = -1
   // Axis.OnlinePtoModeCUEnumValue = PTO（脉冲 A 和方向 B）
   // Axis.OnlinePtoModeCU = 16#0000_0002
   // Axis.SelectedChannel1EnumCU = %Q0.6
   // Pulse.MinDeltaDeltaFrequencyCU = 0.004
   // Pulse.MaxDeltaDeltaFrequencyCU = 1.0E+10
   // Pulse.MinDeltaFrequencyCU = 0.005
   // Pulse.MaxDeltaFrequencyCU = 9.5E+9
   // Pulse.MinFrequencyCU = 1.0
   // Pulse.MaxFrequencyCU = 30000.0
   // Pulse.OutputSourceCU = 16#0000_0000
   // Axis.SelectPTO = 3
   // Axis.OnlinePtoIndexCU = 3
END_DATA_BLOCK

FUNCTION_BLOCK "alarm"   // FB1, LAD
{ S7_Optimized_Access := 'TRUE' }
VERSION : 0.1
   VAR
      "tempI4.4" : Bool;
      "tempI4.5" : Bool;
      "time" : IEC_TIMER;
      time_1 : IEC_TIMER;
      time_2 : IEC_TIMER;
      time_3 : IEC_TIMER;
      time_4 : IEC_TIMER;
      time_5 : IEC_TIMER;
      time_6 : IEC_TIMER;
      time_7 : IEC_TIMER;
      time_8 : IEC_TIMER;
      time_9 : IEC_TIMER;
      IEC_Timer_0_Instance : TON_TIME;
      IEC_Timer_0_Instance_1 : TON_TIME;
   END_VAR
   VAR_TEMP   // added for the SCL form of the ladder/FBD networks
      _w1 : Bool;
      _w2 : Bool;
   END_VAR
BEGIN

REGION Network 1
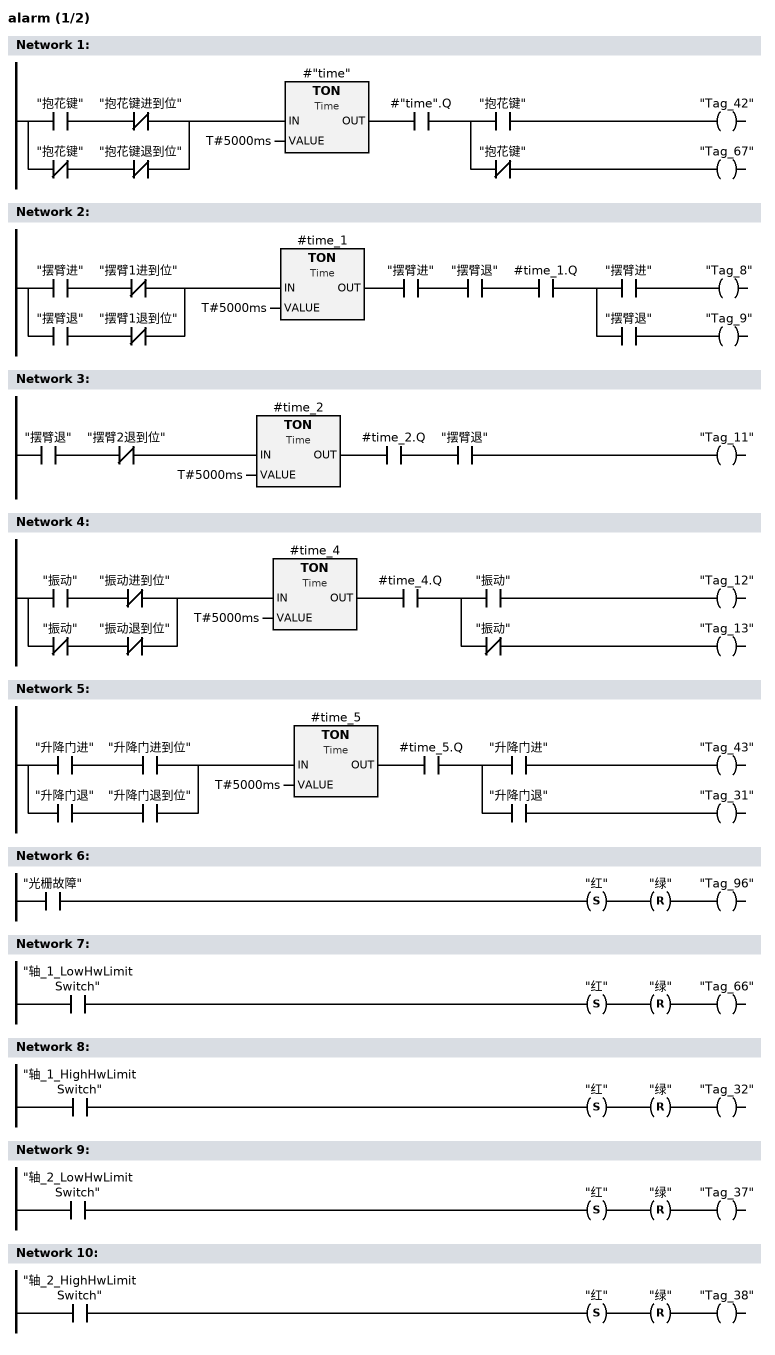
   #_w1 := ("抱花键" AND NOT "抱花键进到位") OR (NOT "抱花键" AND NOT "抱花键退到位");
   #"time".TON(IN := #_w1, PT := T#5000ms);   // TON coil
   #_w2 := #_w1 AND #"time".Q;
   "Tag_42" := #_w2 AND "抱花键";
   "Tag_67" := #_w2 AND NOT "抱花键";
END_REGION

REGION Network 2
   #_w1 := ("摆臂进" AND NOT "摆臂1进到位") OR ("摆臂退" AND NOT "摆臂1退到位");
   #time_1.TON(IN := #_w1, PT := T#5000ms);   // TON coil
   #_w2 := #_w1 AND "摆臂进" AND "摆臂退" AND #time_1.Q;
   "Tag_8" := #_w2 AND "摆臂进";
   "Tag_9" := #_w2 AND "摆臂退";
END_REGION

REGION Network 3
   #_w1 := "摆臂退" AND NOT "摆臂2退到位";
   #time_2.TON(IN := #_w1, PT := T#5000ms);   // TON coil
   "Tag_11" := #_w1 AND #time_2.Q AND "摆臂退";
END_REGION

REGION Network 4
   #_w1 := ("振动" AND NOT "振动进到位") OR (NOT "振动" AND NOT "振动退到位");
   #time_4.TON(IN := #_w1, PT := T#5000ms);   // TON coil
   #_w2 := #_w1 AND #time_4.Q;
   "Tag_12" := #_w2 AND "振动";
   "Tag_13" := #_w2 AND NOT "振动";
END_REGION

REGION Network 5
   #_w1 := ("升降门进" AND "升降门进到位") OR ("升降门退" AND "升降门退到位");
   #time_5.TON(IN := #_w1, PT := T#5000ms);   // TON coil
   #_w2 := #_w1 AND #time_5.Q;
   "Tag_43" := #_w2 AND "升降门进";
   "Tag_31" := #_w2 AND "升降门退";
END_REGION

REGION Network 6
   RUNG wire#powerrail
      Contact( "光栅故障" )
      S_Coil( "红" )
      R_Coil( "绿" )
      Coil( "Tag_96" )
   END_RUNG
   // the same network as SCL:
   IF "光栅故障" THEN
       "红" := TRUE;
       "绿" := FALSE;
   END_IF;
   "Tag_96" := "光栅故障";
END_REGION

REGION Network 7
   RUNG wire#powerrail
      Contact( "轴_1_LowHwLimitSwitch" )
      S_Coil( "红" )
      R_Coil( "绿" )
      Coil( "Tag_66" )
   END_RUNG
   // the same network as SCL:
   IF "轴_1_LowHwLimitSwitch" THEN
       "红" := TRUE;
       "绿" := FALSE;
   END_IF;
   "Tag_66" := "轴_1_LowHwLimitSwitch";
END_REGION

REGION Network 8
   RUNG wire#powerrail
      Contact( "轴_1_HighHwLimitSwitch" )
      S_Coil( "红" )
      R_Coil( "绿" )
      Coil( "Tag_32" )
   END_RUNG
   // the same network as SCL:
   IF "轴_1_HighHwLimitSwitch" THEN
       "红" := TRUE;
       "绿" := FALSE;
   END_IF;
   "Tag_32" := "轴_1_HighHwLimitSwitch";
END_REGION

REGION Network 9
   RUNG wire#powerrail
      Contact( "轴_2_LowHwLimitSwitch" )
      S_Coil( "红" )
      R_Coil( "绿" )
      Coil( "Tag_37" )
   END_RUNG
   // the same network as SCL:
   IF "轴_2_LowHwLimitSwitch" THEN
       "红" := TRUE;
       "绿" := FALSE;
   END_IF;
   "Tag_37" := "轴_2_LowHwLimitSwitch";
END_REGION

REGION Network 10
   RUNG wire#powerrail
      Contact( "轴_2_HighHwLimitSwitch" )
      S_Coil( "红" )
      R_Coil( "绿" )
      Coil( "Tag_38" )
   END_RUNG
   // the same network as SCL:
   IF "轴_2_HighHwLimitSwitch" THEN
       "红" := TRUE;
       "绿" := FALSE;
   END_IF;
   "Tag_38" := "轴_2_HighHwLimitSwitch";
END_REGION

REGION Network 12
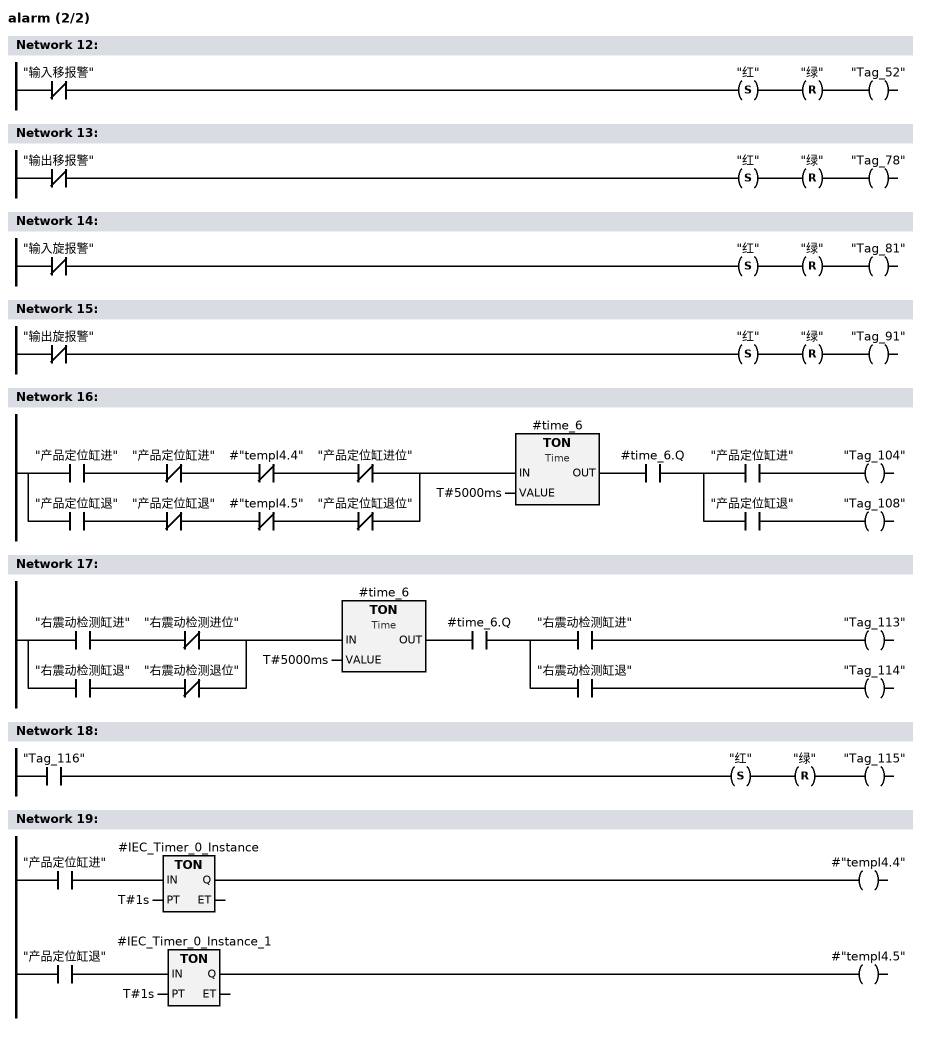
   RUNG wire#powerrail
      I_Contact( "输入移报警" )
      S_Coil( "红" )
      R_Coil( "绿" )
      Coil( "Tag_52" )
   END_RUNG
   // the same network as SCL:
   IF NOT "输入移报警" THEN
       "红" := TRUE;
       "绿" := FALSE;
   END_IF;
   "Tag_52" := NOT "输入移报警";
END_REGION

REGION Network 13
   RUNG wire#powerrail
      I_Contact( "输出移报警" )
      S_Coil( "红" )
      R_Coil( "绿" )
      Coil( "Tag_78" )
   END_RUNG
   // the same network as SCL:
   IF NOT "输出移报警" THEN
       "红" := TRUE;
       "绿" := FALSE;
   END_IF;
   "Tag_78" := NOT "输出移报警";
END_REGION

REGION Network 14
   RUNG wire#powerrail
      I_Contact( "输入旋报警" )
      S_Coil( "红" )
      R_Coil( "绿" )
      Coil( "Tag_81" )
   END_RUNG
   // the same network as SCL:
   IF NOT "输入旋报警" THEN
       "红" := TRUE;
       "绿" := FALSE;
   END_IF;
   "Tag_81" := NOT "输入旋报警";
END_REGION

REGION Network 15
   RUNG wire#powerrail
      I_Contact( "输出旋报警" )
      S_Coil( "红" )
      R_Coil( "绿" )
      Coil( "Tag_91" )
   END_RUNG
   // the same network as SCL:
   IF NOT "输出旋报警" THEN
       "红" := TRUE;
       "绿" := FALSE;
   END_IF;
   "Tag_91" := NOT "输出旋报警";
END_REGION

REGION Network 16
   #_w1 := ("产品定位缸进" AND NOT "产品定位缸进" AND NOT #"tempI4.4" AND NOT "产品定位缸进位") OR ("产品定位缸退" AND NOT "产品定位缸退" AND NOT #"tempI4.5" AND NOT "产品定位缸退位");
   #time_6.TON(IN := #_w1, PT := T#5000ms);   // TON coil
   #_w2 := #_w1 AND #time_6.Q;
   "Tag_104" := #_w2 AND "产品定位缸进";
   "Tag_108" := #_w2 AND "产品定位缸退";
END_REGION

REGION Network 17
   #_w1 := ("右震动检测缸进" AND NOT "右震动检测进位") OR ("右震动检测缸退" AND NOT "右震动检测退位");
   #time_6.TON(IN := #_w1, PT := T#5000ms);   // TON coil
   #_w2 := #_w1 AND #time_6.Q;
   "Tag_113" := #_w2 AND "右震动检测缸进";
   "Tag_114" := #_w2 AND "右震动检测缸退";
END_REGION

REGION Network 18
   RUNG wire#powerrail
      Contact( "Tag_116" )
      S_Coil( "红" )
      R_Coil( "绿" )
      Coil( "Tag_115" )
   END_RUNG
   // the same network as SCL:
   IF "Tag_116" THEN
       "红" := TRUE;
       "绿" := FALSE;
   END_IF;
   "Tag_115" := "Tag_116";
END_REGION

REGION Network 19
   #IEC_Timer_0_Instance(IN := "产品定位缸进", PT := T#1s);   // TON
   #"tempI4.4" := #IEC_Timer_0_Instance.Q;
   #IEC_Timer_0_Instance_1(IN := "产品定位缸退", PT := T#1s);   // TON
   #"tempI4.5" := #IEC_Timer_0_Instance_1.Q;
END_REGION
END_FUNCTION_BLOCK

FUNCTION_BLOCK "reset"   // FB2, LAD
{ S7_Optimized_Access := 'TRUE' }
VERSION : 0.1
   VAR_INPUT
      stt : Bool;
      stp : Bool;
   END_VAR
   VAR_OUTPUT
      done : Bool;
      error : Bool;
      busy : Bool;
   END_VAR
   VAR
      p1 : Real;
      p2 : Real;
      "m" : Array[0..100] of Bool;
      Done_1 : Array[0..5] of Bool;
      "time" : IEC_TIMER;
      IEC_Timer_0_Instance : TON_TIME;
      MC_Reset_Instance : MC_Reset;
      MC_Home_Instance : MC_Home;
      MC_MoveAbsolute_Instance : MC_MoveAbsolute;
      CTRL_HSC_0_Instance : CTRL_HSC;
   END_VAR
   VAR_TEMP
      done1 : Bool;
      done2 : Bool;
      done3 : Bool;
      done4 : Bool;
   END_VAR
   VAR_TEMP   // added for the SCL form of the ladder/FBD networks
      _w1 : Bool;
   END_VAR
BEGIN

REGION Network 1
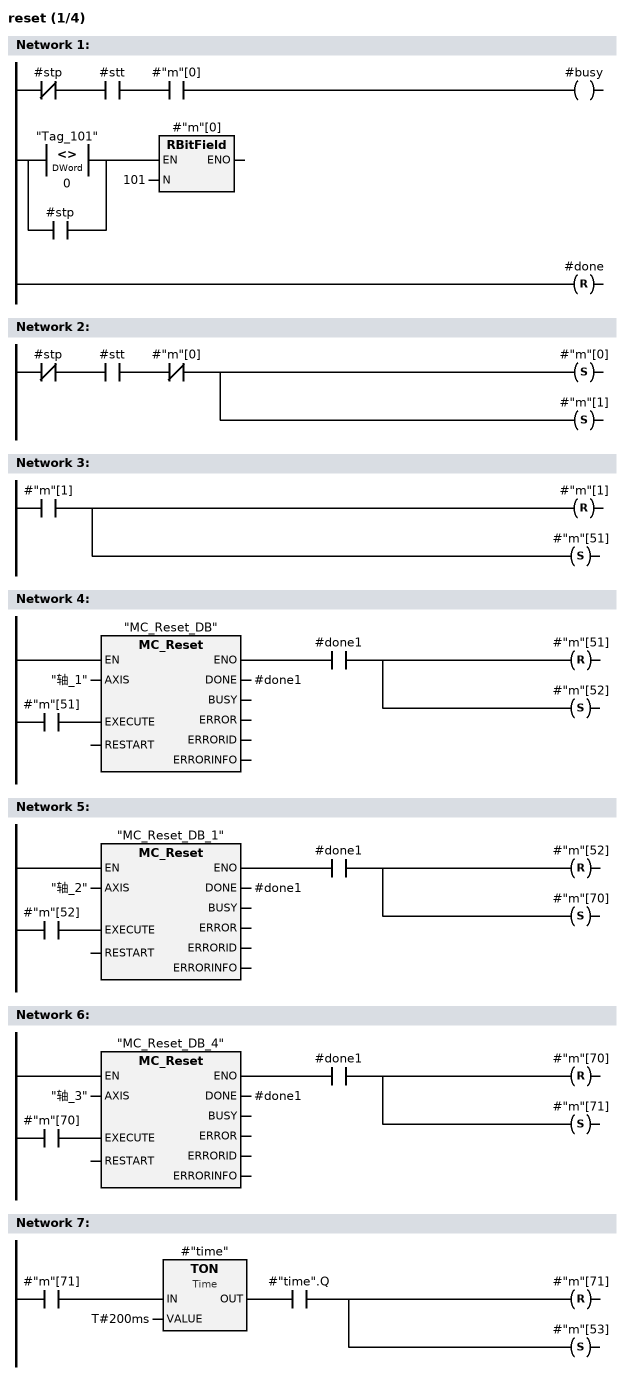
   // no SCL statement known for RBitField: written as a call
   #busy := NOT #stp AND #stt AND #"m"[0];
   IF ("Tag_101" <> 0) OR #stp THEN RBitField(n := 101, operand := #"m"[0]); END_IF;
   #done := FALSE;
END_REGION

REGION Network 2
   RUNG wire#powerrail
      I_Contact( #stp )
      Contact( #stt )
      I_Contact( #"m"[0] )
      wire#w1
      S_Coil( #"m"[0] )
   END_RUNG
   RUNG wire#w1
      S_Coil( #"m"[1] )
   END_RUNG
   // the same network as SCL:
   #_w1 := NOT #stp AND #stt AND NOT #"m"[0];
   IF #_w1 THEN
       #"m"[0] := TRUE;
       #"m"[1] := TRUE;
   END_IF;
END_REGION

REGION Network 3
   RUNG wire#powerrail
      Contact( #"m"[1] )
      wire#w1
      R_Coil( #"m"[1] )
   END_RUNG
   RUNG wire#w1
      S_Coil( #"m"[51] )
   END_RUNG
   // the same network as SCL:
   #_w1 := #"m"[1];
   IF #_w1 THEN
       #"m"[1] := FALSE;
       #"m"[51] := TRUE;
   END_IF;
END_REGION

REGION Network 4
   // ENO of a box is taken as its EN; it also drops when the box reports an error
   "MC_Reset_DB"(Axis := "轴_1", Execute := #"m"[51], Done => #done1);   // MC_Reset
   IF #done1 THEN
       #"m"[51] := FALSE;
       #"m"[52] := TRUE;
   END_IF;
END_REGION

REGION Network 5
   // ENO of a box is taken as its EN; it also drops when the box reports an error
   "MC_Reset_DB_1"(Axis := "轴_2", Execute := #"m"[52], Done => #done1);   // MC_Reset
   IF #done1 THEN
       #"m"[52] := FALSE;
       #"m"[70] := TRUE;
   END_IF;
END_REGION

REGION Network 6
   // ENO of a box is taken as its EN; it also drops when the box reports an error
   "MC_Reset_DB_4"(Axis := "轴_3", Execute := #"m"[70], Done => #done1);   // MC_Reset
   IF #done1 THEN
       #"m"[70] := FALSE;
       #"m"[71] := TRUE;
   END_IF;
END_REGION

REGION Network 7
   #"time".TON(IN := #"m"[71], PT := T#200ms);   // TON coil
   #_w1 := #"m"[71] AND #"time".Q;
   IF #_w1 THEN
       #"m"[71] := FALSE;
       #"m"[53] := TRUE;
   END_IF;
END_REGION

REGION Network 8
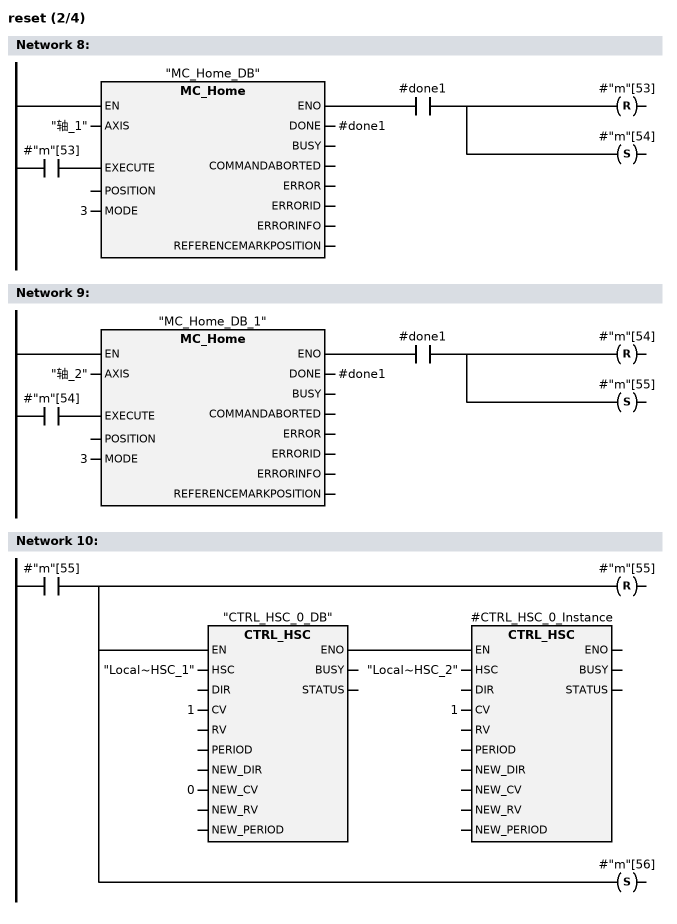
   // ENO of a box is taken as its EN; it also drops when the box reports an error
   "MC_Home_DB"(Axis := "轴_1", Execute := #"m"[53], Mode := 3, Done => #done1);   // MC_Home
   IF #done1 THEN
       #"m"[53] := FALSE;
       #"m"[54] := TRUE;
   END_IF;
END_REGION

REGION Network 9
   // ENO of a box is taken as its EN; it also drops when the box reports an error
   "MC_Home_DB_1"(Axis := "轴_2", Execute := #"m"[54], Mode := 3, Done => #done1);   // MC_Home
   IF #done1 THEN
       #"m"[54] := FALSE;
       #"m"[55] := TRUE;
   END_IF;
END_REGION

REGION Network 10
   // ENO of a box is taken as its EN; it also drops when the box reports an error
   #_w1 := #"m"[55];
   IF #_w1 THEN
       #"m"[55] := FALSE;
       "CTRL_HSC_0_DB"(HSC := "Local~HSC_1", CV := 1, NEW_CV := 0);   // CTRL_HSC
       #CTRL_HSC_0_Instance(HSC := "Local~HSC_2", CV := 1);   // CTRL_HSC
       #"m"[56] := TRUE;
   END_IF;
END_REGION

REGION Network 11
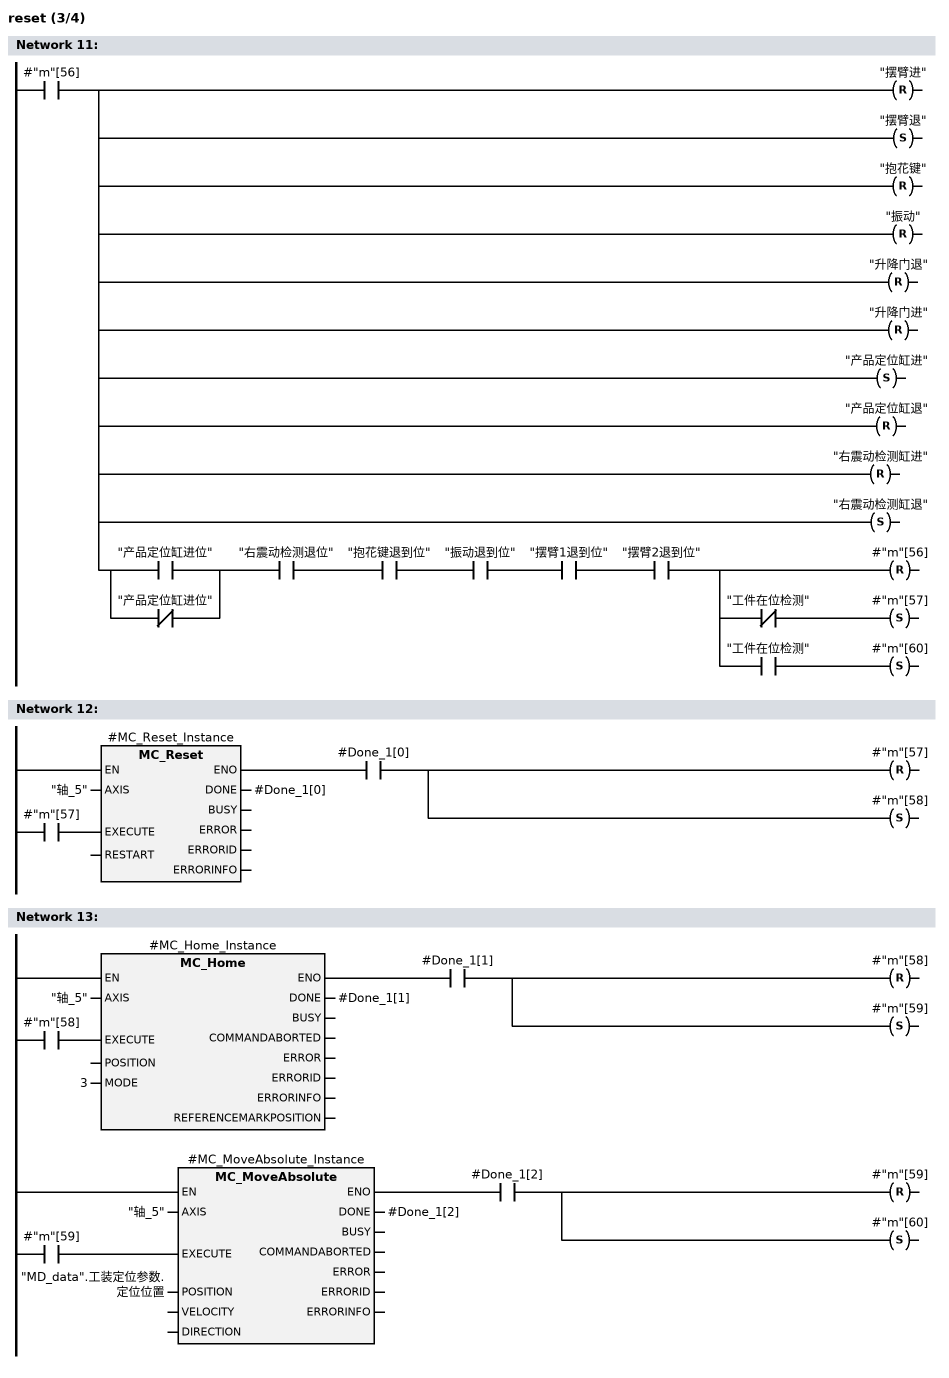
   RUNG wire#powerrail
      Contact( #"m"[56] )
      wire#w1
      R_Coil( "摆臂进" )
   END_RUNG
   RUNG wire#w1
      S_Coil( "摆臂退" )
   END_RUNG
   RUNG wire#w1
      R_Coil( "抱花键" )
   END_RUNG
   RUNG wire#w1
      R_Coil( "振动" )
   END_RUNG
   RUNG wire#w1
      R_Coil( "升降门退" )
   END_RUNG
   RUNG wire#w1
      R_Coil( "升降门进" )
   END_RUNG
   RUNG wire#w1
      S_Coil( "产品定位缸进" )
   END_RUNG
   RUNG wire#w1
      R_Coil( "产品定位缸退" )
   END_RUNG
   RUNG wire#w1
      R_Coil( "右震动检测缸进" )
   END_RUNG
   RUNG wire#w1
      S_Coil( "右震动检测缸退" )
   END_RUNG
   RUNG wire#w1
      Contact( "产品定位缸进位" )
      wire#w2
      Contact( "右震动检测退位" )
      Contact( "抱花键退到位" )
      Contact( "振动退到位" )
      Contact( "摆臂1退到位" )
      Contact( "摆臂2退到位" )
      wire#w3
      R_Coil( #"m"[56] )
   END_RUNG
   RUNG wire#w1
      I_Contact( "产品定位缸进位" )
   END_RUNG wire#w2
   RUNG wire#w3
      I_Contact( "工件在位检测" )
      S_Coil( #"m"[57] )
   END_RUNG
   RUNG wire#w3
      Contact( "工件在位检测" )
      S_Coil( #"m"[60] )
   END_RUNG
   // the same network as SCL:
   IF #"m"[56] THEN
       "摆臂进" := FALSE;
       "摆臂退" := TRUE;
       "抱花键" := FALSE;
       "振动" := FALSE;
       "升降门退" := FALSE;
       "升降门进" := FALSE;
       "产品定位缸进" := TRUE;
       "产品定位缸退" := FALSE;
       "右震动检测缸进" := FALSE;
       "右震动检测缸退" := TRUE;
   END_IF;
   #_w1 := #"m"[56] AND ("产品定位缸进位" OR NOT "产品定位缸进位") AND "右震动检测退位" AND "抱花键退到位" AND "振动退到位" AND "摆臂1退到位" AND "摆臂2退到位";
   IF #_w1 THEN #"m"[56] := FALSE; END_IF;
   IF #_w1 AND NOT "工件在位检测" THEN #"m"[57] := TRUE; END_IF;
   IF #_w1 AND "工件在位检测" THEN #"m"[60] := TRUE; END_IF;
END_REGION

REGION Network 12
   // ENO of a box is taken as its EN; it also drops when the box reports an error
   #MC_Reset_Instance(Axis := "轴_5", Execute := #"m"[57], Done => #Done_1[0]);   // MC_Reset
   IF #Done_1[0] THEN
       #"m"[57] := FALSE;
       #"m"[58] := TRUE;
   END_IF;
END_REGION

REGION Network 13
   // ENO of a box is taken as its EN; it also drops when the box reports an error
   #MC_Home_Instance(Axis := "轴_5", Execute := #"m"[58], Mode := 3, Done => #Done_1[1]);   // MC_Home
   IF #Done_1[1] THEN
       #"m"[58] := FALSE;
       #"m"[59] := TRUE;
   END_IF;
   #MC_MoveAbsolute_Instance(Axis := "轴_5",   // MC_MoveAbsolute
                           Execute := #"m"[59],
                           Position := "MD_data".工装定位参数.定位位置,
                           Done => #Done_1[2]);
   IF #Done_1[2] THEN
       #"m"[59] := FALSE;
       #"m"[60] := TRUE;
   END_IF;
END_REGION

REGION Network 14
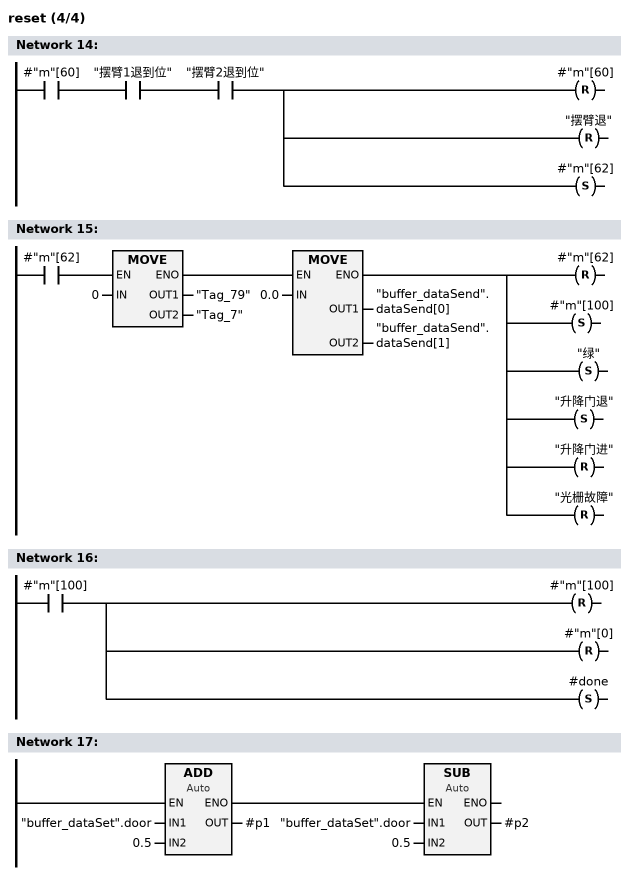
   RUNG wire#powerrail
      Contact( #"m"[60] )
      Contact( "摆臂1退到位" )
      Contact( "摆臂2退到位" )
      wire#w1
      R_Coil( #"m"[60] )
   END_RUNG
   RUNG wire#w1
      R_Coil( "摆臂退" )
   END_RUNG
   RUNG wire#w1
      S_Coil( #"m"[62] )
   END_RUNG
   // the same network as SCL:
   #_w1 := #"m"[60] AND "摆臂1退到位" AND "摆臂2退到位";
   IF #_w1 THEN
       #"m"[60] := FALSE;
       "摆臂退" := FALSE;
       #"m"[62] := TRUE;
   END_IF;
END_REGION

REGION Network 15
   RUNG wire#powerrail
      Contact( #"m"[62] )
      Move(in := 0, out1 => "Tag_79", out2 => "Tag_7")
      Move(in := 0.0, out1 => "buffer_dataSend".dataSend[0], out2 => "buffer_dataSend".dataSend[1])
      wire#w1
      R_Coil( #"m"[62] )
   END_RUNG
   RUNG wire#w1
      S_Coil( #"m"[100] )
   END_RUNG
   RUNG wire#w1
      S_Coil( "绿" )
   END_RUNG
   RUNG wire#w1
      S_Coil( "升降门退" )
   END_RUNG
   RUNG wire#w1
      R_Coil( "升降门进" )
   END_RUNG
   RUNG wire#w1
      R_Coil( "光栅故障" )
   END_RUNG
   // the same network as SCL:
   IF #"m"[62] THEN
       "Tag_79" := 0;
       "Tag_7" := 0;
       "buffer_dataSend".dataSend[0] := 0.0;
       "buffer_dataSend".dataSend[1] := 0.0;
   END_IF;
   #_w1 := #"m"[62];
   IF #_w1 THEN
       #"m"[62] := FALSE;
       #"m"[100] := TRUE;
       "绿" := TRUE;
       "升降门退" := TRUE;
       "升降门进" := FALSE;
       "光栅故障" := FALSE;
   END_IF;
END_REGION

REGION Network 16
   RUNG wire#powerrail
      Contact( #"m"[100] )
      wire#w1
      R_Coil( #"m"[100] )
   END_RUNG
   RUNG wire#w1
      R_Coil( #"m"[0] )
   END_RUNG
   RUNG wire#w1
      S_Coil( #done )
   END_RUNG
   // the same network as SCL:
   #_w1 := #"m"[100];
   IF #_w1 THEN
       #"m"[100] := FALSE;
       #"m"[0] := FALSE;
       #done := TRUE;
   END_IF;
END_REGION

REGION Network 17
   RUNG wire#powerrail
      Add(in1 := "buffer_dataSet".door, in2 := 0.5, out => #p1)
      Sub(in1 := "buffer_dataSet".door, in2 := 0.5, out => #p2)
   END_RUNG
   // the same network as SCL:
   #p1 := "buffer_dataSet".door + 0.5;
   #p2 := "buffer_dataSet".door - 0.5;
END_REGION
END_FUNCTION_BLOCK

FUNCTION_BLOCK "manual"   // FB3, LAD
{ S7_Optimized_Access := 'TRUE' }
VERSION : 0.1
   VAR_INPUT
      open : Bool;
      emg : Bool;
   END_VAR
   VAR
      temp_1 : Bool;
      temp_2 : Bool;
      buffer : Array[0..20] of Byte;
      emg_n : Bool;
      MC_MoveJog_Instance : MC_MoveJog;
      MC_Reset_Instance : MC_Reset;
      MC_Power_Instance : MC_Power;
      MC_Home_Instance : MC_Home;
      MC_MoveAbsolute_Instance : MC_MoveAbsolute;
      MC_Power_Instance_1 : MC_Power;
      IEC_Timer_0_Instance : TON_TIME;
      IEC_Timer_0_Instance_1 : TON_TIME;
      IEC_Timer_0_Instance_2 : TON_TIME;
      IEC_Timer_0_Instance_3 : TON_TIME;
      IEC_Timer_0_Instance_4 : TON_TIME;
      IEC_Timer_0_Instance_5 : TON_TIME;
      MC_Halt_Instance : MC_Halt;
   END_VAR
   VAR_TEMP
      "m" : Real;
      m_1 : Real;
   END_VAR
   VAR_TEMP   // added for the SCL form of the ladder/FBD networks
      _w1 : Bool;
      _w2 : Bool;
      _w3 : Bool;
      _w4 : Bool;
   END_VAR
BEGIN

REGION Network 2
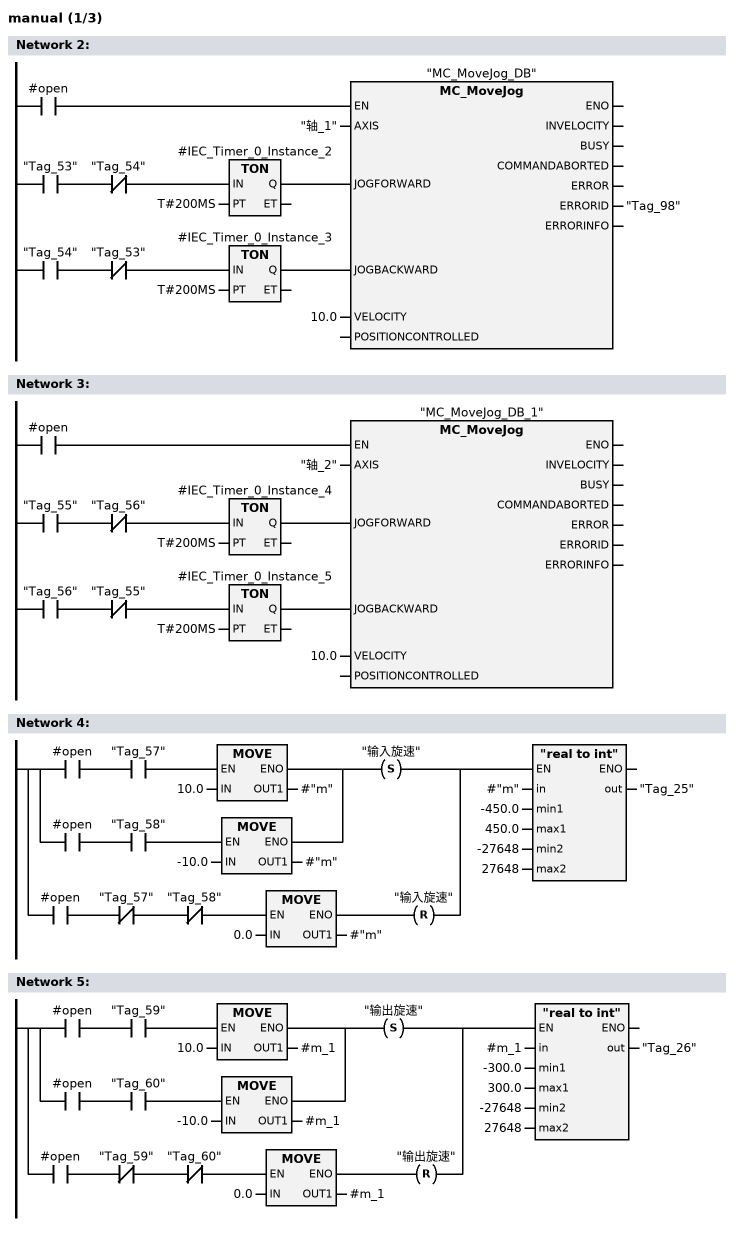
   #IEC_Timer_0_Instance_2(IN := "Tag_53" AND NOT "Tag_54", PT := T#200MS);   // TON
   #IEC_Timer_0_Instance_3(IN := "Tag_54" AND NOT "Tag_53", PT := T#200MS);   // TON
   IF #open THEN
       "MC_MoveJog_DB"(Axis := "轴_1",   // MC_MoveJog
                       JogForward := #IEC_Timer_0_Instance_2.Q,
                       JogBackward := #IEC_Timer_0_Instance_3.Q,
                       Velocity := 10.0,
                       ErrorID => "Tag_98");
   END_IF;
END_REGION

REGION Network 3
   #IEC_Timer_0_Instance_4(IN := "Tag_55" AND NOT "Tag_56", PT := T#200MS);   // TON
   #IEC_Timer_0_Instance_5(IN := "Tag_56" AND NOT "Tag_55", PT := T#200MS);   // TON
   IF #open THEN
       "MC_MoveJog_DB_1"(Axis := "轴_2",   // MC_MoveJog
                         JogForward := #IEC_Timer_0_Instance_4.Q,
                         JogBackward := #IEC_Timer_0_Instance_5.Q,
                         Velocity := 10.0);
   END_IF;
END_REGION

REGION Network 4
   RUNG wire#powerrail
      Contact( #open )
      Contact( "Tag_57" )
      Move(in := 10.0, out1 => #"m")
      wire#w1
      S_Coil( "输入旋速" )
      wire#w2
      "real to int"(in := #"m", min1 := -450.0, max1 := 450.0, min2 := -27648, max2 := 27648, out => "Tag_25")
   END_RUNG
   RUNG wire#powerrail
      Contact( #open )
      Contact( "Tag_58" )
      Move(in := -10.0, out1 => #"m")
   END_RUNG wire#w1
   RUNG wire#powerrail
      Contact( #open )
      I_Contact( "Tag_57" )
      I_Contact( "Tag_58" )
      Move(in := 0.0, out1 => #"m")
      R_Coil( "输入旋速" )
   END_RUNG wire#w2
   // the same network as SCL:
   #_w1 := #open AND "Tag_57";
   IF #_w1 THEN #"m" := 10.0; END_IF;
   #_w2 := #open AND "Tag_58";
   IF #_w2 THEN #"m" := -10.0; END_IF;
   #_w3 := #_w1 OR #_w2;
   IF #_w3 THEN "输入旋速" := TRUE; END_IF;
   #_w4 := #open AND NOT "Tag_57" AND NOT "Tag_58";
   IF #_w4 THEN
       #"m" := 0.0;
       "输入旋速" := FALSE;
   END_IF;
   IF #_w3 OR #_w4 THEN
       "real to int"(in := #"m", min1 := -450.0, max1 := 450.0, min2 := -27648, max2 := 27648, out => "Tag_25");
   END_IF;
END_REGION

REGION Network 5
   RUNG wire#powerrail
      Contact( #open )
      Contact( "Tag_59" )
      Move(in := 10.0, out1 => #m_1)
      wire#w1
      S_Coil( "输出旋速" )
      wire#w2
      "real to int"(in := #m_1, min1 := -300.0, max1 := 300.0, min2 := -27648, max2 := 27648, out => "Tag_26")
   END_RUNG
   RUNG wire#powerrail
      Contact( #open )
      Contact( "Tag_60" )
      Move(in := -10.0, out1 => #m_1)
   END_RUNG wire#w1
   RUNG wire#powerrail
      Contact( #open )
      I_Contact( "Tag_59" )
      I_Contact( "Tag_60" )
      Move(in := 0.0, out1 => #m_1)
      R_Coil( "输出旋速" )
   END_RUNG wire#w2
   // the same network as SCL:
   #_w1 := #open AND "Tag_59";
   IF #_w1 THEN #m_1 := 10.0; END_IF;
   #_w2 := #open AND "Tag_60";
   IF #_w2 THEN #m_1 := -10.0; END_IF;
   #_w3 := #_w1 OR #_w2;
   IF #_w3 THEN "输出旋速" := TRUE; END_IF;
   #_w4 := #open AND NOT "Tag_59" AND NOT "Tag_60";
   IF #_w4 THEN
       #m_1 := 0.0;
       "输出旋速" := FALSE;
   END_IF;
   IF #_w3 OR #_w4 THEN
       "real to int"(in := #m_1, min1 := -300.0, max1 := 300.0, min2 := -27648, max2 := 27648, out => "Tag_26");
   END_IF;
END_REGION

REGION Network 6
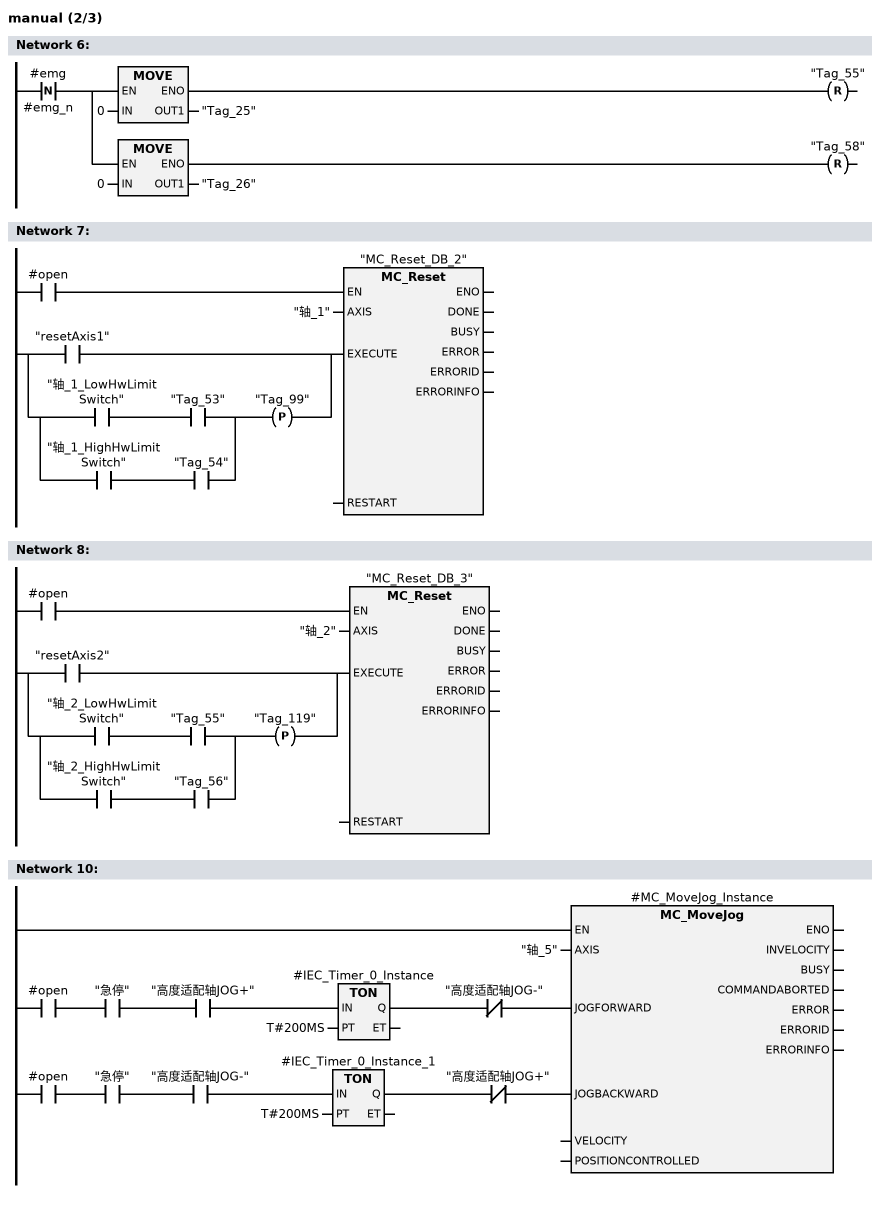
   RUNG wire#powerrail
      N_Contact(operand := #emg, bit := #emg_n)
      wire#w1
      Move(in := 0, out1 => "Tag_25")
      R_Coil( "Tag_55" )
   END_RUNG
   RUNG wire#w1
      Move(in := 0, out1 => "Tag_26")
      R_Coil( "Tag_58" )
   END_RUNG
   // the same network as SCL:
   #_w1 := NOT #emg AND #emg_n;   // falling edge of #emg
   #emg_n := #emg;
   IF #_w1 THEN
       "Tag_25" := 0;
       "Tag_55" := FALSE;
       "Tag_26" := 0;
       "Tag_58" := FALSE;
   END_IF;
END_REGION

REGION Network 7
   #_w1 := ("轴_1_LowHwLimitSwitch" AND "Tag_53") OR ("轴_1_HighHwLimitSwitch" AND "Tag_54");
   #_w2 := #_w1 AND NOT "Tag_99";   // rising edge
   "Tag_99" := #_w1;
   IF #open THEN
       "MC_Reset_DB_2"(Axis := "轴_1", Execute := "resetAxis1" OR #_w2);   // MC_Reset
   END_IF;
END_REGION

REGION Network 8
   #_w1 := ("轴_2_LowHwLimitSwitch" AND "Tag_55") OR ("轴_2_HighHwLimitSwitch" AND "Tag_56");
   #_w2 := #_w1 AND NOT "Tag_119";   // rising edge
   "Tag_119" := #_w1;
   IF #open THEN
       "MC_Reset_DB_3"(Axis := "轴_2", Execute := "resetAxis2" OR #_w2);   // MC_Reset
   END_IF;
END_REGION

REGION Network 10
   #IEC_Timer_0_Instance(IN := #open AND "急停" AND "高度适配轴JOG+", PT := T#200MS);   // TON
   #IEC_Timer_0_Instance_1(IN := #open AND "急停" AND "高度适配轴JOG-", PT := T#200MS);   // TON
   #MC_MoveJog_Instance(Axis := "轴_5",   // MC_MoveJog
                        JogForward := #IEC_Timer_0_Instance.Q AND NOT "高度适配轴JOG-",
                        JogBackward := #IEC_Timer_0_Instance_1.Q AND NOT "高度适配轴JOG+");
END_REGION

REGION Network 11
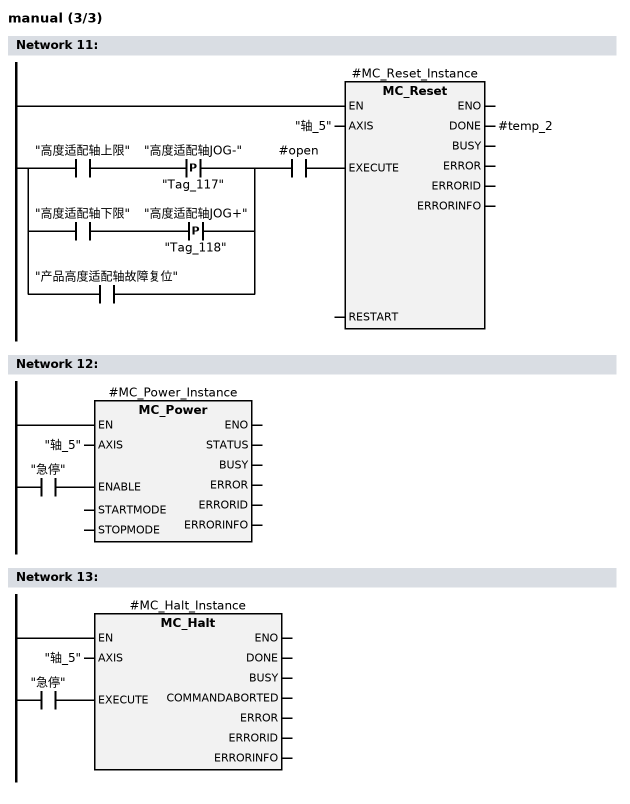
   #_w1 := "高度适配轴上限" AND "高度适配轴JOG-" AND NOT "Tag_117";   // rising edge of "高度适配轴JOG-"
   "Tag_117" := "高度适配轴JOG-";
   #_w2 := "高度适配轴下限" AND "高度适配轴JOG+" AND NOT "Tag_118";   // rising edge of "高度适配轴JOG+"
   "Tag_118" := "高度适配轴JOG+";
   #MC_Reset_Instance(Axis := "轴_5", Execute := (#_w1 OR #_w2 OR "产品高度适配轴故障复位") AND #open, Done => #temp_2);   // MC_Reset
END_REGION

REGION Network 12
   #MC_Power_Instance(Axis := "轴_5", Enable := "急停");   // MC_Power
END_REGION

REGION Network 13
   #MC_Halt_Instance(Axis := "轴_5", Execute := "急停");   // MC_Halt
END_REGION
END_FUNCTION_BLOCK

FUNCTION_BLOCK "套输入轴花键"   // FB4, LAD
{ S7_Optimized_Access := 'TRUE' }
VERSION : 0.1
   VAR_INPUT
      stt : Bool;
      stp : Bool;
   END_VAR
   VAR_OUTPUT
      done : Bool;
      error : Bool;
      busy : Bool;
   END_VAR
   VAR
      "m" : Array[0..100] of Bool;
      "time" : IEC_TIMER;
      time_1 : IEC_TIMER;
      speedC : Real;
   END_VAR
   VAR_TEMP
      done1 : Bool;
      done2 : Bool;
      done3 : Bool;
      done4 : Bool;
      n : Bool;
      n_1 : Bool;
      lang : Real;
   END_VAR
   VAR_TEMP   // added for the SCL form of the ladder/FBD networks
      _w1 : Bool;
      _w2 : Bool;
   END_VAR
BEGIN

REGION Network 1
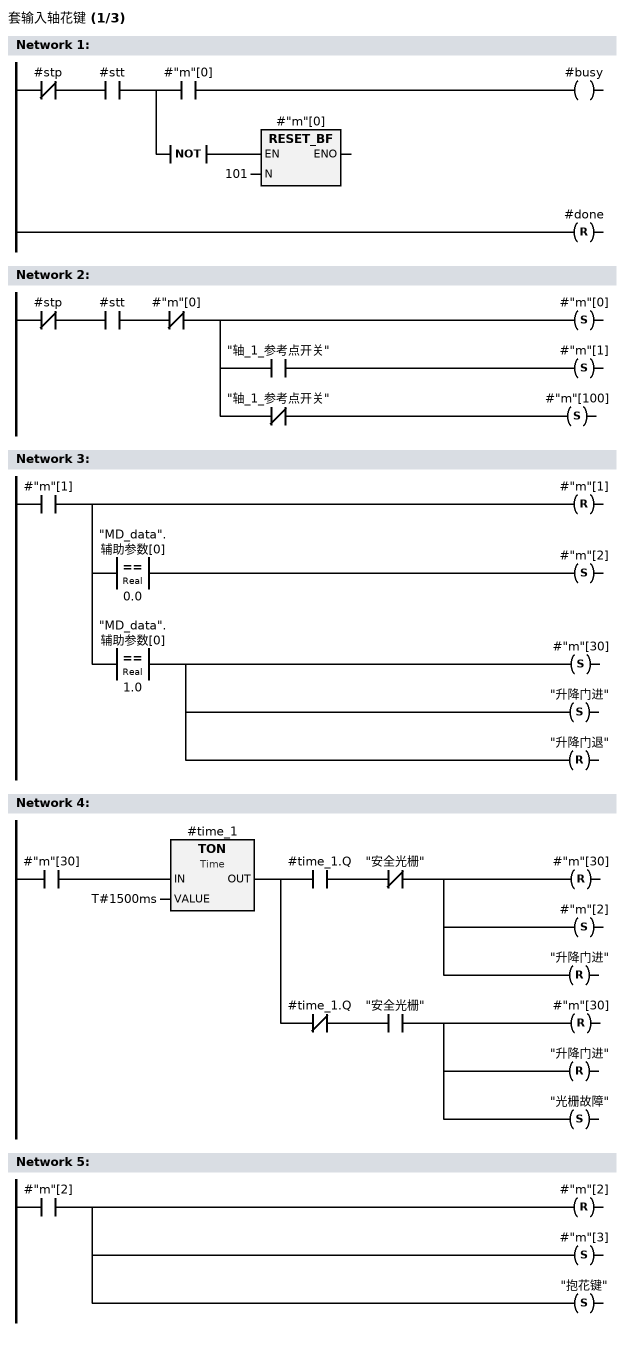
   // no SCL statement known for RBitfield: written as a call
   #_w1 := NOT #stp AND #stt;
   #busy := #_w1 AND #"m"[0];
   IF NOT #_w1 THEN RESET_BF(operand := #"m"[0], n := 101); END_IF;
   #done := FALSE;
END_REGION

REGION Network 2
   RUNG wire#powerrail
      I_Contact( #stp )
      Contact( #stt )
      I_Contact( #"m"[0] )
      wire#w1
      S_Coil( #"m"[0] )
   END_RUNG
   RUNG wire#w1
      Contact( "轴_1_参考点开关" )
      S_Coil( #"m"[1] )
   END_RUNG
   RUNG wire#w1
      I_Contact( "轴_1_参考点开关" )
      S_Coil( #"m"[100] )
   END_RUNG
   // the same network as SCL:
   #_w1 := NOT #stp AND #stt AND NOT #"m"[0];
   IF #_w1 THEN #"m"[0] := TRUE; END_IF;
   IF #_w1 AND "轴_1_参考点开关" THEN #"m"[1] := TRUE; END_IF;
   IF #_w1 AND NOT "轴_1_参考点开关" THEN #"m"[100] := TRUE; END_IF;
END_REGION

REGION Network 3
   RUNG wire#powerrail
      Contact( #"m"[1] )
      wire#w1
      R_Coil( #"m"[1] )
   END_RUNG
   RUNG wire#w1
      { S7_Templates := "SrcType := Real" } EQ_Contact(in1 := "MD_data".辅助参数[0], in2 := 0.0)
      S_Coil( #"m"[2] )
   END_RUNG
   RUNG wire#w1
      { S7_Templates := "SrcType := Real" } EQ_Contact(in1 := "MD_data".辅助参数[0], in2 := 1.0)
      wire#w2
      S_Coil( #"m"[30] )
   END_RUNG
   RUNG wire#w2
      S_Coil( "升降门进" )
   END_RUNG
   RUNG wire#w2
      R_Coil( "升降门退" )
   END_RUNG
   // the same network as SCL:
   #_w1 := #"m"[1];
   IF #_w1 THEN #"m"[1] := FALSE; END_IF;
   IF #_w1 AND ("MD_data".辅助参数[0] = 0.0) THEN #"m"[2] := TRUE; END_IF;
   IF #_w1 AND ("MD_data".辅助参数[0] = 1.0) THEN
       #"m"[30] := TRUE;
       "升降门进" := TRUE;
       "升降门退" := FALSE;
   END_IF;
END_REGION

REGION Network 4
   #time_1.TON(IN := #"m"[30], PT := T#1500ms);   // TON coil
   #_w1 := #"m"[30];
   #_w2 := #"m"[30] AND #time_1.Q AND NOT "安全光栅";
   IF #_w2 THEN
       #"m"[30] := FALSE;
       #"m"[2] := TRUE;
       "升降门进" := FALSE;
   END_IF;
   IF #_w1 AND NOT #time_1.Q AND "安全光栅" THEN
       #"m"[30] := FALSE;
       "升降门进" := FALSE;
       "光栅故障" := TRUE;
   END_IF;
END_REGION

REGION Network 5
   RUNG wire#powerrail
      Contact( #"m"[2] )
      wire#w1
      R_Coil( #"m"[2] )
   END_RUNG
   RUNG wire#w1
      S_Coil( #"m"[3] )
   END_RUNG
   RUNG wire#w1
      S_Coil( "抱花键" )
   END_RUNG
   // the same network as SCL:
   #_w1 := #"m"[2];
   IF #_w1 THEN
       #"m"[2] := FALSE;
       #"m"[3] := TRUE;
       "抱花键" := TRUE;
   END_IF;
END_REGION

REGION Network 6
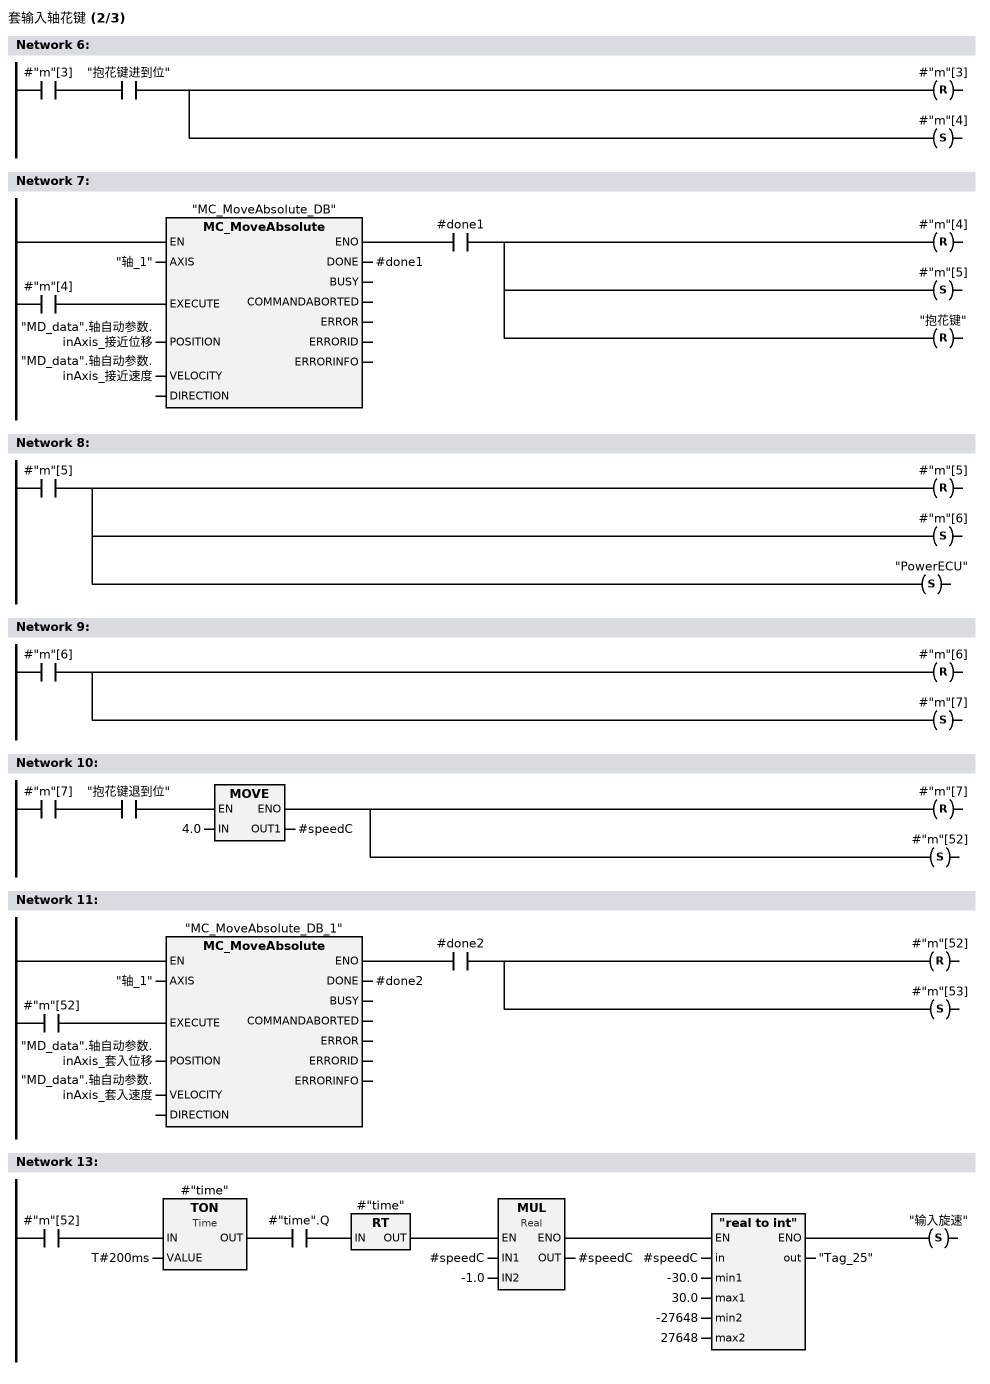
   RUNG wire#powerrail
      Contact( #"m"[3] )
      Contact( "抱花键进到位" )
      wire#w1
      R_Coil( #"m"[3] )
   END_RUNG
   RUNG wire#w1
      S_Coil( #"m"[4] )
   END_RUNG
   // the same network as SCL:
   #_w1 := #"m"[3] AND "抱花键进到位";
   IF #_w1 THEN
       #"m"[3] := FALSE;
       #"m"[4] := TRUE;
   END_IF;
END_REGION

REGION Network 7
   // ENO of a box is taken as its EN; it also drops when the box reports an error
   "MC_MoveAbsolute_DB"(Axis := "轴_1",   // MC_MoveAbsolute
                        Execute := #"m"[4],
                        Position := "MD_data".轴自动参数.inAxis_接近位移,
                        Velocity := "MD_data".轴自动参数.inAxis_接近速度,
                        Done => #done1);
   IF #done1 THEN
       #"m"[4] := FALSE;
       #"m"[5] := TRUE;
       "抱花键" := FALSE;
   END_IF;
END_REGION

REGION Network 8
   RUNG wire#powerrail
      Contact( #"m"[5] )
      wire#w1
      R_Coil( #"m"[5] )
   END_RUNG
   RUNG wire#w1
      S_Coil( #"m"[6] )
   END_RUNG
   RUNG wire#w1
      S_Coil( "PowerECU" )
   END_RUNG
   // the same network as SCL:
   #_w1 := #"m"[5];
   IF #_w1 THEN
       #"m"[5] := FALSE;
       #"m"[6] := TRUE;
       "PowerECU" := TRUE;
   END_IF;
END_REGION

REGION Network 9
   RUNG wire#powerrail
      Contact( #"m"[6] )
      wire#w1
      R_Coil( #"m"[6] )
   END_RUNG
   RUNG wire#w1
      S_Coil( #"m"[7] )
   END_RUNG
   // the same network as SCL:
   #_w1 := #"m"[6];
   IF #_w1 THEN
       #"m"[6] := FALSE;
       #"m"[7] := TRUE;
   END_IF;
END_REGION

REGION Network 10
   RUNG wire#powerrail
      Contact( #"m"[7] )
      Contact( "抱花键退到位" )
      Move(in := 4.0, out1 => #speedC)
      wire#w1
      R_Coil( #"m"[7] )
   END_RUNG
   RUNG wire#w1
      S_Coil( #"m"[52] )
   END_RUNG
   // the same network as SCL:
   IF #"m"[7] AND "抱花键退到位" THEN #speedC := 4.0; END_IF;
   #_w1 := #"m"[7] AND "抱花键退到位";
   IF #_w1 THEN
       #"m"[7] := FALSE;
       #"m"[52] := TRUE;
   END_IF;
END_REGION

REGION Network 11
   // ENO of a box is taken as its EN; it also drops when the box reports an error
   "MC_MoveAbsolute_DB_1"(Axis := "轴_1",   // MC_MoveAbsolute
                          Execute := #"m"[52],
                          Position := "MD_data".轴自动参数.inAxis_套入位移,
                          Velocity := "MD_data".轴自动参数.inAxis_套入速度,
                          Done => #done2);
   IF #done2 THEN
       #"m"[52] := FALSE;
       #"m"[53] := TRUE;
   END_IF;
END_REGION

REGION Network 13
   #"time".TON(IN := #"m"[52], PT := T#200ms);   // TON coil
   #_w1 := #"m"[52] AND #"time".Q;
   IF #_w1 THEN
       RESET_TIMER(#"time");
       #speedC := #speedC * (-1.0);
   END_IF;
   "real to int"(EN := #_w1,
                 in := #speedC,
                 min1 := -30.0,
                 max1 := 30.0,
                 min2 := -27648,
                 max2 := 27648,
                 out => "Tag_25",
                 ENO => #_w2);
   IF #_w2 THEN "输入旋速" := TRUE; END_IF;
END_REGION

REGION Network 14
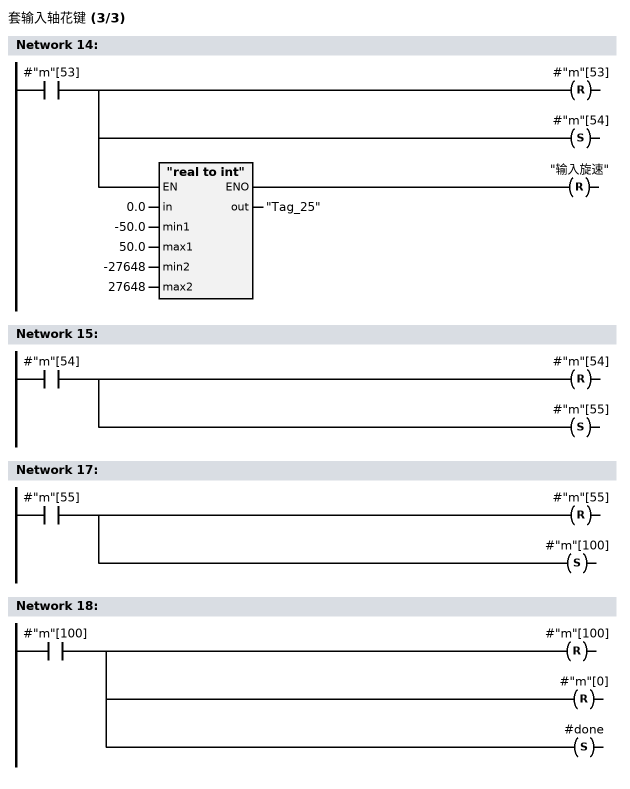
   RUNG wire#powerrail
      Contact( #"m"[53] )
      wire#w1
      R_Coil( #"m"[53] )
   END_RUNG
   RUNG wire#w1
      S_Coil( #"m"[54] )
   END_RUNG
   RUNG wire#w1
      "real to int"(in := 0.0, min1 := -50.0, max1 := 50.0, min2 := -27648, max2 := 27648, out => "Tag_25")
      R_Coil( "输入旋速" )
   END_RUNG
   // the same network as SCL:
   #_w1 := #"m"[53];
   IF #_w1 THEN
       #"m"[53] := FALSE;
       #"m"[54] := TRUE;
   END_IF;
   "real to int"(EN := #_w1,
                 in := 0.0,
                 min1 := -50.0,
                 max1 := 50.0,
                 min2 := -27648,
                 max2 := 27648,
                 out => "Tag_25",
                 ENO => #_w2);
   IF #_w2 THEN "输入旋速" := FALSE; END_IF;
END_REGION

REGION Network 15
   RUNG wire#powerrail
      Contact( #"m"[54] )
      wire#w1
      R_Coil( #"m"[54] )
   END_RUNG
   RUNG wire#w1
      S_Coil( #"m"[55] )
   END_RUNG
   // the same network as SCL:
   #_w1 := #"m"[54];
   IF #_w1 THEN
       #"m"[54] := FALSE;
       #"m"[55] := TRUE;
   END_IF;
END_REGION

REGION Network 17
   RUNG wire#powerrail
      Contact( #"m"[55] )
      wire#w1
      R_Coil( #"m"[55] )
   END_RUNG
   RUNG wire#w1
      S_Coil( #"m"[100] )
   END_RUNG
   // the same network as SCL:
   #_w1 := #"m"[55];
   IF #_w1 THEN
       #"m"[55] := FALSE;
       #"m"[100] := TRUE;
   END_IF;
END_REGION

REGION Network 18
   RUNG wire#powerrail
      Contact( #"m"[100] )
      wire#w1
      R_Coil( #"m"[100] )
   END_RUNG
   RUNG wire#w1
      R_Coil( #"m"[0] )
   END_RUNG
   RUNG wire#w1
      S_Coil( #done )
   END_RUNG
   // the same network as SCL:
   #_w1 := #"m"[100];
   IF #_w1 THEN
       #"m"[100] := FALSE;
       #"m"[0] := FALSE;
       #done := TRUE;
   END_IF;
END_REGION
END_FUNCTION_BLOCK

FUNCTION_BLOCK "套输出轴花键"   // FB5, LAD
{ S7_Optimized_Access := 'TRUE' }
VERSION : 0.1
   VAR_INPUT
      stt : Bool;
      stp : Bool;
   END_VAR
   VAR_OUTPUT
      done : Bool;
      error : Bool;
      busy : Bool;
   END_VAR
   VAR
      "m" : Array[0..100] of Bool;
      "time" : IEC_TIMER;
      time_1 : IEC_TIMER;
      speedC : Real;
      MC_MoveAbsolute_Instance : MC_MoveAbsolute;
   END_VAR
   VAR_TEMP
      done1 : Bool;
      done2 : Bool;
      done3 : Bool;
      done4 : Bool;
      timeset : Time;
      n : Bool;
      n_1 : Bool;
      lang : Real;
   END_VAR
   VAR_TEMP   // added for the SCL form of the ladder/FBD networks
      _w1 : Bool;
      _w2 : Bool;
   END_VAR
BEGIN

REGION Network 1
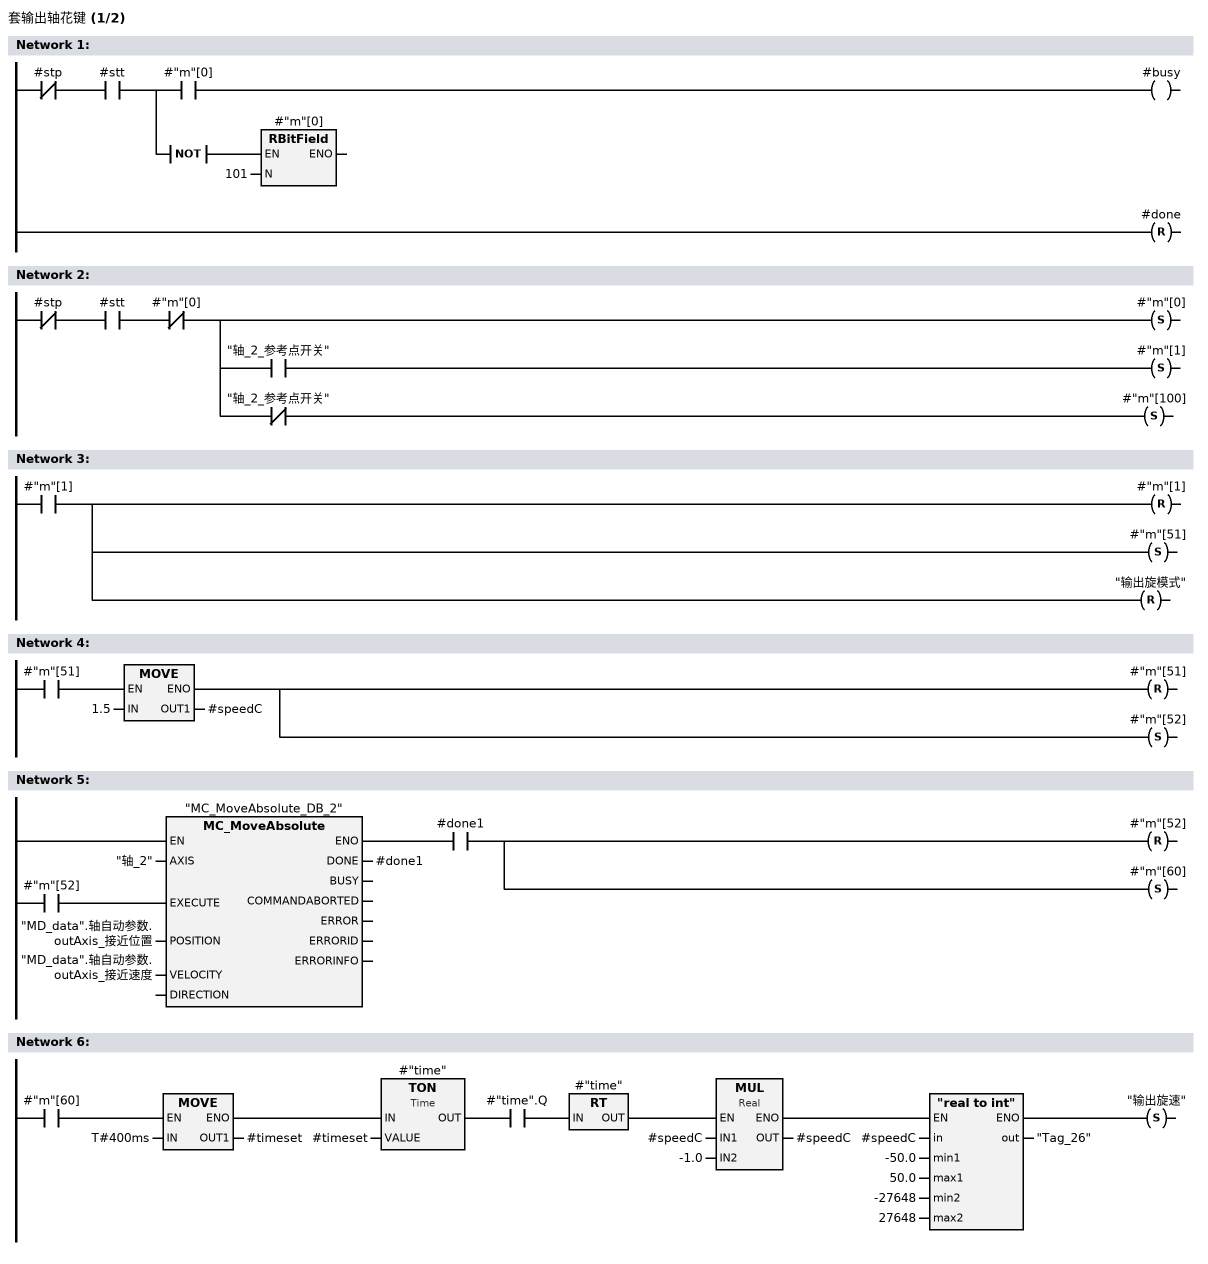
   // no SCL statement known for RBitField: written as a call
   #_w1 := NOT #stp AND #stt;
   #busy := #_w1 AND #"m"[0];
   IF NOT #_w1 THEN RBitField(n := 101, operand := #"m"[0]); END_IF;
   #done := FALSE;
END_REGION

REGION Network 2
   RUNG wire#powerrail
      I_Contact( #stp )
      Contact( #stt )
      I_Contact( #"m"[0] )
      wire#w1
      S_Coil( #"m"[0] )
   END_RUNG
   RUNG wire#w1
      Contact( "轴_2_参考点开关" )
      S_Coil( #"m"[1] )
   END_RUNG
   RUNG wire#w1
      I_Contact( "轴_2_参考点开关" )
      S_Coil( #"m"[100] )
   END_RUNG
   // the same network as SCL:
   #_w1 := NOT #stp AND #stt AND NOT #"m"[0];
   IF #_w1 THEN #"m"[0] := TRUE; END_IF;
   IF #_w1 AND "轴_2_参考点开关" THEN #"m"[1] := TRUE; END_IF;
   IF #_w1 AND NOT "轴_2_参考点开关" THEN #"m"[100] := TRUE; END_IF;
END_REGION

REGION Network 3
   RUNG wire#powerrail
      Contact( #"m"[1] )
      wire#w1
      R_Coil( #"m"[1] )
   END_RUNG
   RUNG wire#w1
      S_Coil( #"m"[51] )
   END_RUNG
   RUNG wire#w1
      R_Coil( "输出旋模式" )
   END_RUNG
   // the same network as SCL:
   #_w1 := #"m"[1];
   IF #_w1 THEN
       #"m"[1] := FALSE;
       #"m"[51] := TRUE;
       "输出旋模式" := FALSE;
   END_IF;
END_REGION

REGION Network 4
   RUNG wire#powerrail
      Contact( #"m"[51] )
      Move(in := 1.5, out1 => #speedC)
      wire#w1
      R_Coil( #"m"[51] )
   END_RUNG
   RUNG wire#w1
      S_Coil( #"m"[52] )
   END_RUNG
   // the same network as SCL:
   IF #"m"[51] THEN #speedC := 1.5; END_IF;
   #_w1 := #"m"[51];
   IF #_w1 THEN
       #"m"[51] := FALSE;
       #"m"[52] := TRUE;
   END_IF;
END_REGION

REGION Network 5
   // ENO of a box is taken as its EN; it also drops when the box reports an error
   "MC_MoveAbsolute_DB_2"(Axis := "轴_2",   // MC_MoveAbsolute
                          Execute := #"m"[52],
                          Position := "MD_data".轴自动参数.outAxis_接近位置,
                          Velocity := "MD_data".轴自动参数.outAxis_接近速度,
                          Done => #done1);
   IF #done1 THEN
       #"m"[52] := FALSE;
       #"m"[60] := TRUE;
   END_IF;
END_REGION

REGION Network 6
   IF #"m"[60] THEN #timeset := T#400ms; END_IF;
   #"time".TON(IN := #"m"[60], PT := #timeset);   // TON coil
   #_w1 := #"m"[60] AND #"time".Q;
   IF #_w1 THEN
       RESET_TIMER(#"time");
       #speedC := #speedC * (-1.0);
   END_IF;
   "real to int"(EN := #_w1,
                 in := #speedC,
                 min1 := -50.0,
                 max1 := 50.0,
                 min2 := -27648,
                 max2 := 27648,
                 out => "Tag_26",
                 ENO => #_w2);
   IF #_w2 THEN "输出旋速" := TRUE; END_IF;
END_REGION

REGION Network 7
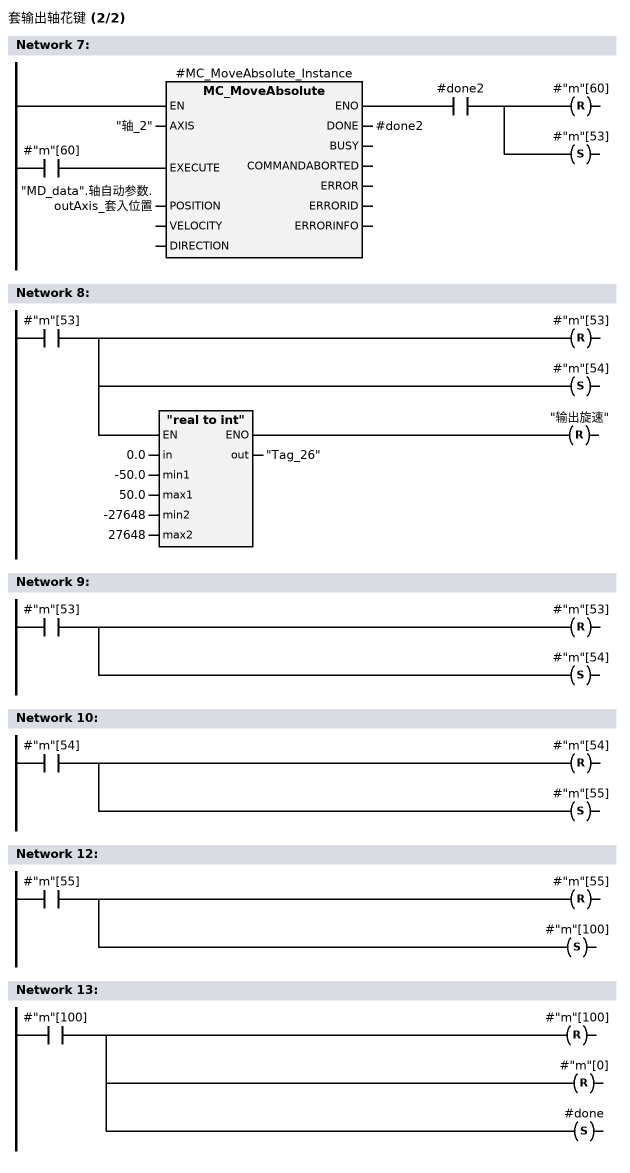
   // ENO of a box is taken as its EN; it also drops when the box reports an error
   #MC_MoveAbsolute_Instance(Axis := "轴_2",   // MC_MoveAbsolute
                           Execute := #"m"[60],
                           Position := "MD_data".轴自动参数.outAxis_套入位置,
                           Done => #done2);
   IF #done2 THEN
       #"m"[60] := FALSE;
       #"m"[53] := TRUE;
   END_IF;
END_REGION

REGION Network 8
   RUNG wire#powerrail
      Contact( #"m"[53] )
      wire#w1
      R_Coil( #"m"[53] )
   END_RUNG
   RUNG wire#w1
      S_Coil( #"m"[54] )
   END_RUNG
   RUNG wire#w1
      "real to int"(in := 0.0, min1 := -50.0, max1 := 50.0, min2 := -27648, max2 := 27648, out => "Tag_26")
      R_Coil( "输出旋速" )
   END_RUNG
   // the same network as SCL:
   #_w1 := #"m"[53];
   IF #_w1 THEN
       #"m"[53] := FALSE;
       #"m"[54] := TRUE;
   END_IF;
   "real to int"(EN := #_w1,
                 in := 0.0,
                 min1 := -50.0,
                 max1 := 50.0,
                 min2 := -27648,
                 max2 := 27648,
                 out => "Tag_26",
                 ENO => #_w2);
   IF #_w2 THEN "输出旋速" := FALSE; END_IF;
END_REGION

REGION Network 9
   RUNG wire#powerrail
      Contact( #"m"[53] )
      wire#w1
      R_Coil( #"m"[53] )
   END_RUNG
   RUNG wire#w1
      S_Coil( #"m"[54] )
   END_RUNG
   // the same network as SCL:
   #_w1 := #"m"[53];
   IF #_w1 THEN
       #"m"[53] := FALSE;
       #"m"[54] := TRUE;
   END_IF;
END_REGION

REGION Network 10
   RUNG wire#powerrail
      Contact( #"m"[54] )
      wire#w1
      R_Coil( #"m"[54] )
   END_RUNG
   RUNG wire#w1
      S_Coil( #"m"[55] )
   END_RUNG
   // the same network as SCL:
   #_w1 := #"m"[54];
   IF #_w1 THEN
       #"m"[54] := FALSE;
       #"m"[55] := TRUE;
   END_IF;
END_REGION

REGION Network 12
   RUNG wire#powerrail
      Contact( #"m"[55] )
      wire#w1
      R_Coil( #"m"[55] )
   END_RUNG
   RUNG wire#w1
      S_Coil( #"m"[100] )
   END_RUNG
   // the same network as SCL:
   #_w1 := #"m"[55];
   IF #_w1 THEN
       #"m"[55] := FALSE;
       #"m"[100] := TRUE;
   END_IF;
END_REGION

REGION Network 13
   RUNG wire#powerrail
      Contact( #"m"[100] )
      wire#w1
      R_Coil( #"m"[100] )
   END_RUNG
   RUNG wire#w1
      R_Coil( #"m"[0] )
   END_RUNG
   RUNG wire#w1
      S_Coil( #done )
   END_RUNG
   // the same network as SCL:
   #_w1 := #"m"[100];
   IF #_w1 THEN
       #"m"[100] := FALSE;
       #"m"[0] := FALSE;
       #done := TRUE;
   END_IF;
END_REGION
END_FUNCTION_BLOCK

FUNCTION_BLOCK "motor_m"   // FB6, LAD
{ S7_Optimized_Access := 'TRUE' }
VERSION : 0.1
   VAR_INPUT
      run : Bool;
      speed : Real;
   END_VAR
   VAR_OUTPUT
      open : Bool;
      value : Int;
   END_VAR
   VAR_TEMP
      "m" : Real;
   END_VAR
BEGIN

REGION Network 1
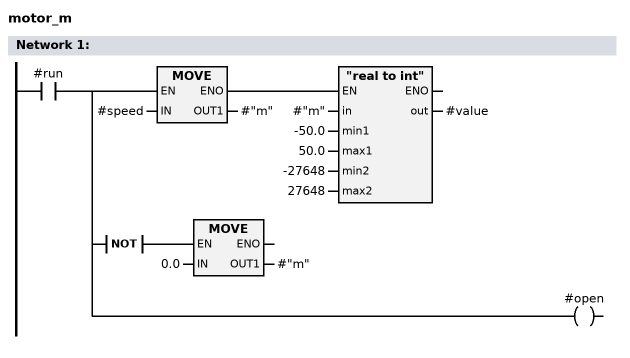
   RUNG wire#powerrail
      Contact( #run )
      wire#w1
      Move(in := #speed, out1 => #"m")
      "real to int"(in := #"m", min1 := -50.0, max1 := 50.0, min2 := -27648, max2 := 27648, out => #value)
   END_RUNG
   RUNG wire#w1
      Not()
      Move(in := 0.0, out1 => #"m")
   END_RUNG
   RUNG wire#w1
      Coil( #open )
   END_RUNG
   // the same network as SCL:
   IF #run THEN
       #"m" := #speed;
       "real to int"(in := #"m", min1 := -50.0, max1 := 50.0, min2 := -27648, max2 := 27648, out => #value);
   END_IF;
   IF NOT #run THEN #"m" := 0.0; END_IF;
   #open := #run;
END_REGION
END_FUNCTION_BLOCK

FUNCTION_BLOCK "空载与标定"   // FB7, LAD
{ S7_Optimized_Access := 'TRUE' }
VERSION : 0.1
   VAR_INPUT
      stt : Bool;
      stp : Bool;
      direction : Bool;
      speed : Real;
      angle : Real;
   END_VAR
   VAR_OUTPUT
      done : Bool;
      error : Bool;
      busy : Bool;
   END_VAR
   VAR
      "m" : Array[0..100] of Bool;
      "time" : IEC_TIMER;
      newCV : DInt;
      angleSet : Real;
      speedSet : Real;
      angleRead : Real;
   END_VAR
   VAR_TEMP   // added for the SCL form of the ladder/FBD networks
      _w1 : Bool;
      _w2 : Bool;
   END_VAR
BEGIN

REGION Network 1
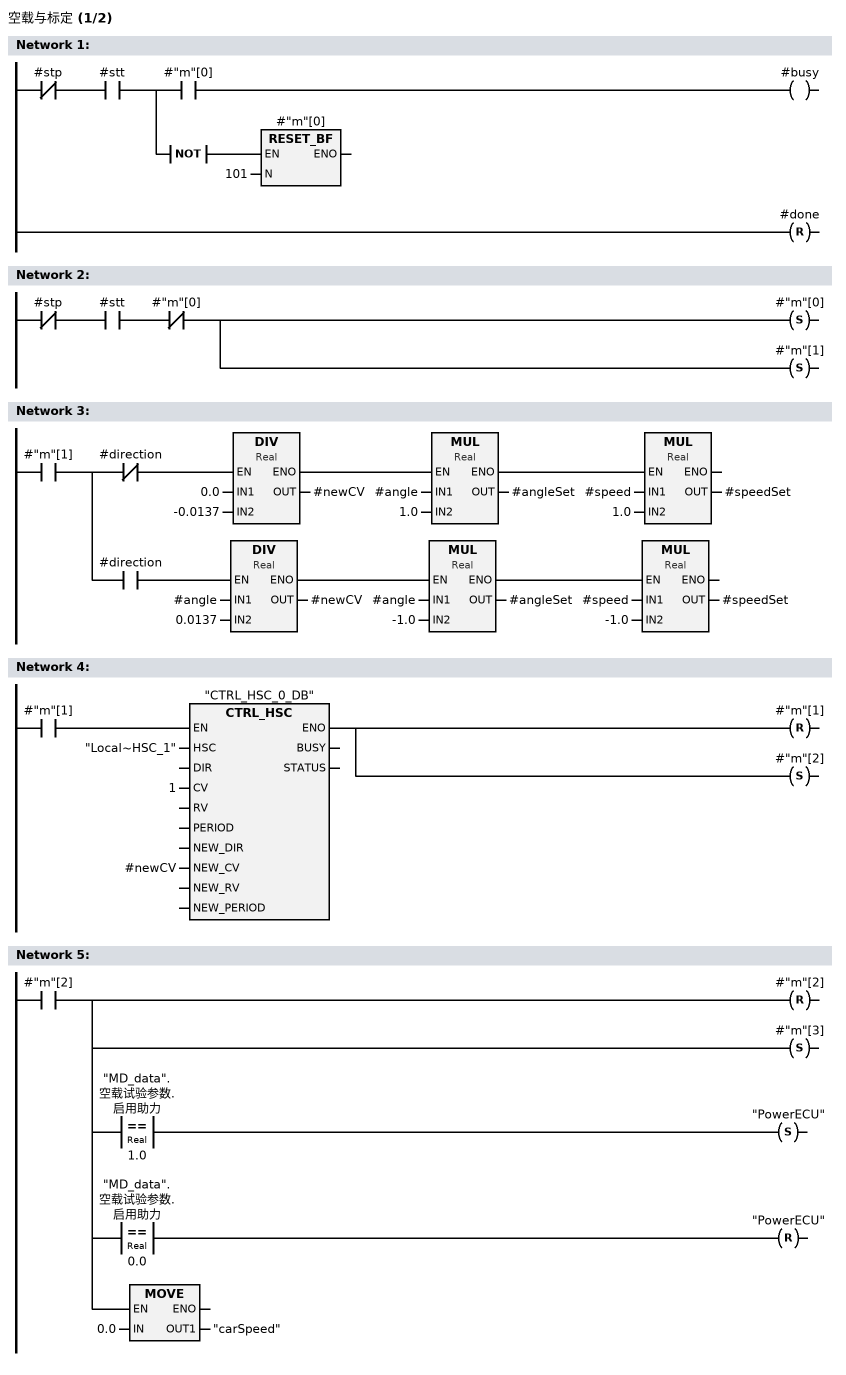
   // no SCL statement known for RBitfield: written as a call
   #_w1 := NOT #stp AND #stt;
   #busy := #_w1 AND #"m"[0];
   IF NOT #_w1 THEN RESET_BF(operand := #"m"[0], n := 101); END_IF;
   #done := FALSE;
END_REGION

REGION Network 2
   RUNG wire#powerrail
      I_Contact( #stp )
      Contact( #stt )
      I_Contact( #"m"[0] )
      wire#w1
      S_Coil( #"m"[0] )
   END_RUNG
   RUNG wire#w1
      S_Coil( #"m"[1] )
   END_RUNG
   // the same network as SCL:
   #_w1 := NOT #stp AND #stt AND NOT #"m"[0];
   IF #_w1 THEN
       #"m"[0] := TRUE;
       #"m"[1] := TRUE;
   END_IF;
END_REGION

REGION Network 3
   RUNG wire#powerrail
      Contact( #"m"[1] )
      wire#w1
      I_Contact( #direction )
      { S7_Templates := "SrcType := Real" } Div(in1 := 0.0, in2 := -0.0137, out => #newCV)
      { S7_Templates := "SrcType := Real" } Mul(in1 := #angle, in2 := 1.0, out => #angleSet)
      { S7_Templates := "SrcType := Real" } Mul(in1 := #speed, in2 := 1.0, out => #speedSet)
   END_RUNG
   RUNG wire#w1
      Contact( #direction )
      { S7_Templates := "SrcType := Real" } Div(in1 := #angle, in2 := 0.0137, out => #newCV)
      { S7_Templates := "SrcType := Real" } Mul(in1 := #angle, in2 := -1.0, out => #angleSet)
      { S7_Templates := "SrcType := Real" } Mul(in1 := #speed, in2 := -1.0, out => #speedSet)
   END_RUNG
   // the same network as SCL:
   IF #"m"[1] AND NOT #direction THEN
       #newCV := 0.0 / (-0.0137);
       #angleSet := #angle * 1.0;
       #speedSet := #speed * 1.0;
   END_IF;
   IF #"m"[1] AND #direction THEN
       #newCV := #angle / 0.0137;
       #angleSet := #angle * (-1.0);
       #speedSet := #speed * (-1.0);
   END_IF;
END_REGION

REGION Network 4
   // ENO of a box is taken as its EN; it also drops when the box reports an error
   IF #"m"[1] THEN
       "CTRL_HSC_0_DB"(HSC := "Local~HSC_1", CV := 1, NEW_CV := #newCV);   // CTRL_HSC
   END_IF;
   #_w1 := #"m"[1];
   IF #_w1 THEN
       #"m"[1] := FALSE;
       #"m"[2] := TRUE;
   END_IF;
END_REGION

REGION Network 5
   RUNG wire#powerrail
      Contact( #"m"[2] )
      wire#w1
      R_Coil( #"m"[2] )
   END_RUNG
   RUNG wire#w1
      S_Coil( #"m"[3] )
   END_RUNG
   RUNG wire#w1
      { S7_Templates := "SrcType := Real" } EQ_Contact(in1 := "MD_data".空载试验参数.启用助力, in2 := 1.0)
      S_Coil( "PowerECU" )
   END_RUNG
   RUNG wire#w1
      { S7_Templates := "SrcType := Real" } EQ_Contact(in1 := "MD_data".空载试验参数.启用助力, in2 := 0.0)
      R_Coil( "PowerECU" )
   END_RUNG
   RUNG wire#w1
      Move(in := 0.0, out1 => "carSpeed")
   END_RUNG
   // the same network as SCL:
   #_w1 := #"m"[2];
   IF #_w1 THEN
       #"m"[2] := FALSE;
       #"m"[3] := TRUE;
   END_IF;
   IF #_w1 AND ("MD_data".空载试验参数.启用助力 = 1.0) THEN "PowerECU" := TRUE; END_IF;
   IF #_w1 AND ("MD_data".空载试验参数.启用助力 = 0.0) THEN "PowerECU" := FALSE; END_IF;
   IF #_w1 THEN "carSpeed" := 0.0; END_IF;
END_REGION

REGION Network 6
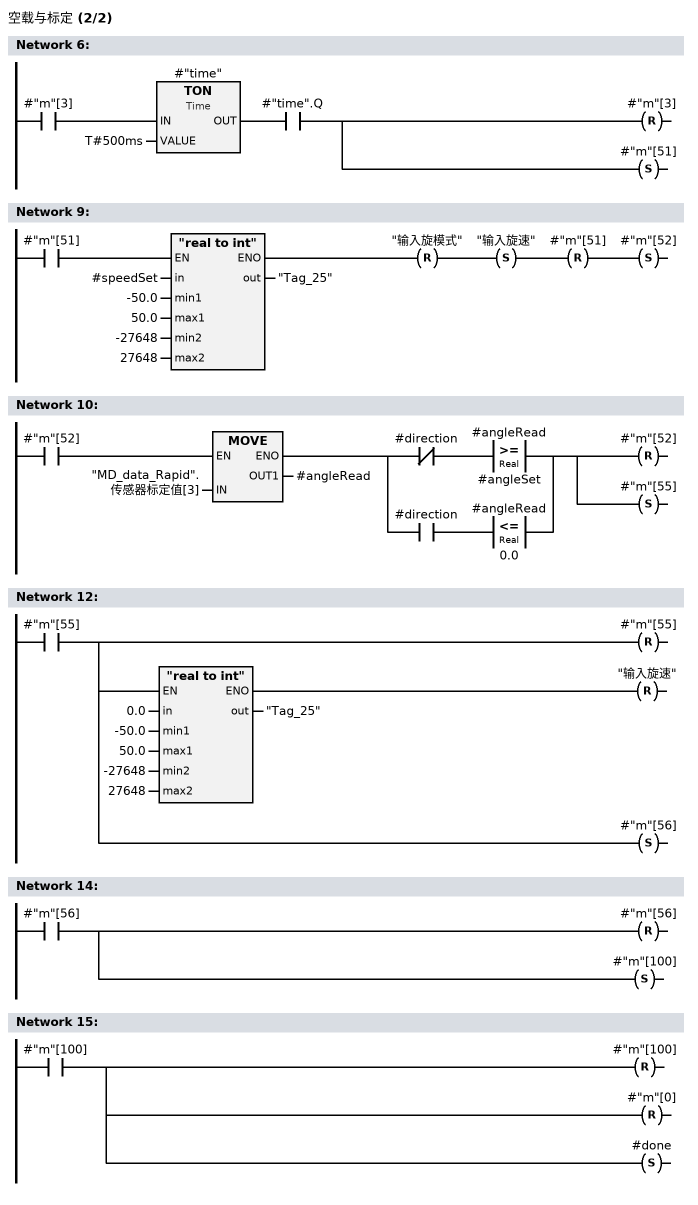
   #"time".TON(IN := #"m"[3], PT := T#500ms);   // TON coil
   #_w1 := #"m"[3] AND #"time".Q;
   IF #_w1 THEN
       #"m"[3] := FALSE;
       #"m"[51] := TRUE;
   END_IF;
END_REGION

REGION Network 9
   RUNG wire#powerrail
      Contact( #"m"[51] )
      "real to int"(in := #speedSet, min1 := -50.0, max1 := 50.0, min2 := -27648, max2 := 27648, out => "Tag_25")
      R_Coil( "输入旋模式" )
      S_Coil( "输入旋速" )
      R_Coil( #"m"[51] )
      S_Coil( #"m"[52] )
   END_RUNG
   // the same network as SCL:
   "real to int"(EN := #"m"[51],
                 in := #speedSet,
                 min1 := -50.0,
                 max1 := 50.0,
                 min2 := -27648,
                 max2 := 27648,
                 out => "Tag_25",
                 ENO => #_w1);
   IF #_w1 THEN
       "输入旋模式" := FALSE;
       "输入旋速" := TRUE;
       #"m"[51] := FALSE;
       #"m"[52] := TRUE;
   END_IF;
END_REGION

REGION Network 10
   RUNG wire#powerrail
      Contact( #"m"[52] )
      Move(in := "MD_data_Rapid".传感器标定值[3], out1 => #angleRead)
      wire#w1
      I_Contact( #direction )
      { S7_Templates := "SrcType := Real" } GE_Contact(in1 := #angleRead, in2 := #angleSet)
      wire#w2
      R_Coil( #"m"[52] )
   END_RUNG
   RUNG wire#w1
      Contact( #direction )
      { S7_Templates := "SrcType := Real" } LE_Contact(in1 := #angleRead, in2 := 0.0)
   END_RUNG wire#w2
   RUNG wire#w2
      S_Coil( #"m"[55] )
   END_RUNG
   // the same network as SCL:
   IF #"m"[52] THEN #angleRead := "MD_data_Rapid".传感器标定值[3]; END_IF;
   #_w1 := #"m"[52] AND ((NOT #direction AND (#angleRead >= #angleSet)) OR (#direction AND (#angleRead <= 0.0)));
   IF #_w1 THEN
       #"m"[52] := FALSE;
       #"m"[55] := TRUE;
   END_IF;
END_REGION

REGION Network 12
   RUNG wire#powerrail
      Contact( #"m"[55] )
      wire#w1
      R_Coil( #"m"[55] )
   END_RUNG
   RUNG wire#w1
      "real to int"(in := 0.0, min1 := -50.0, max1 := 50.0, min2 := -27648, max2 := 27648, out => "Tag_25")
      R_Coil( "输入旋速" )
   END_RUNG
   RUNG wire#w1
      S_Coil( #"m"[56] )
   END_RUNG
   // the same network as SCL:
   #_w1 := #"m"[55];
   IF #_w1 THEN #"m"[55] := FALSE; END_IF;
   "real to int"(EN := #_w1,
                 in := 0.0,
                 min1 := -50.0,
                 max1 := 50.0,
                 min2 := -27648,
                 max2 := 27648,
                 out => "Tag_25",
                 ENO => #_w2);
   IF #_w2 THEN "输入旋速" := FALSE; END_IF;
   IF #_w1 THEN #"m"[56] := TRUE; END_IF;
END_REGION

REGION Network 14
   RUNG wire#powerrail
      Contact( #"m"[56] )
      wire#w1
      R_Coil( #"m"[56] )
   END_RUNG
   RUNG wire#w1
      S_Coil( #"m"[100] )
   END_RUNG
   // the same network as SCL:
   #_w1 := #"m"[56];
   IF #_w1 THEN
       #"m"[56] := FALSE;
       #"m"[100] := TRUE;
   END_IF;
END_REGION

REGION Network 15
   RUNG wire#powerrail
      Contact( #"m"[100] )
      wire#w1
      R_Coil( #"m"[100] )
   END_RUNG
   RUNG wire#w1
      R_Coil( #"m"[0] )
   END_RUNG
   RUNG wire#w1
      S_Coil( #done )
   END_RUNG
   // the same network as SCL:
   #_w1 := #"m"[100];
   IF #_w1 THEN
       #"m"[100] := FALSE;
       #"m"[0] := FALSE;
       #done := TRUE;
   END_IF;
END_REGION
END_FUNCTION_BLOCK

FUNCTION_BLOCK "力特性"   // FB9, LAD
{ S7_Optimized_Access := 'TRUE' }
VERSION : 0.1
   VAR_INPUT
      stt : Bool;
      stp : Bool;
      direction : Bool;
      speed : Real;
      torque : Real;
      load : Real;
   END_VAR
   VAR_OUTPUT
      done : Bool;
      error : Bool;
      busy : Bool;
   END_VAR
   VAR
      "m" : Array[0..100] of Bool;
      "time" : IEC_TIMER;
      speedSet : Real;
      torqueSet : Real;
      IEC_Timer_0_Instance : TON_TIME;
      IEC_Timer_0_Instance_1 : TON_TIME;
   END_VAR
   VAR_TEMP
      torqueTemp : Real;
   END_VAR
   VAR_TEMP   // added for the SCL form of the ladder/FBD networks
      _w1 : Bool;
      _w2 : Bool;
   END_VAR
BEGIN

REGION Network 1
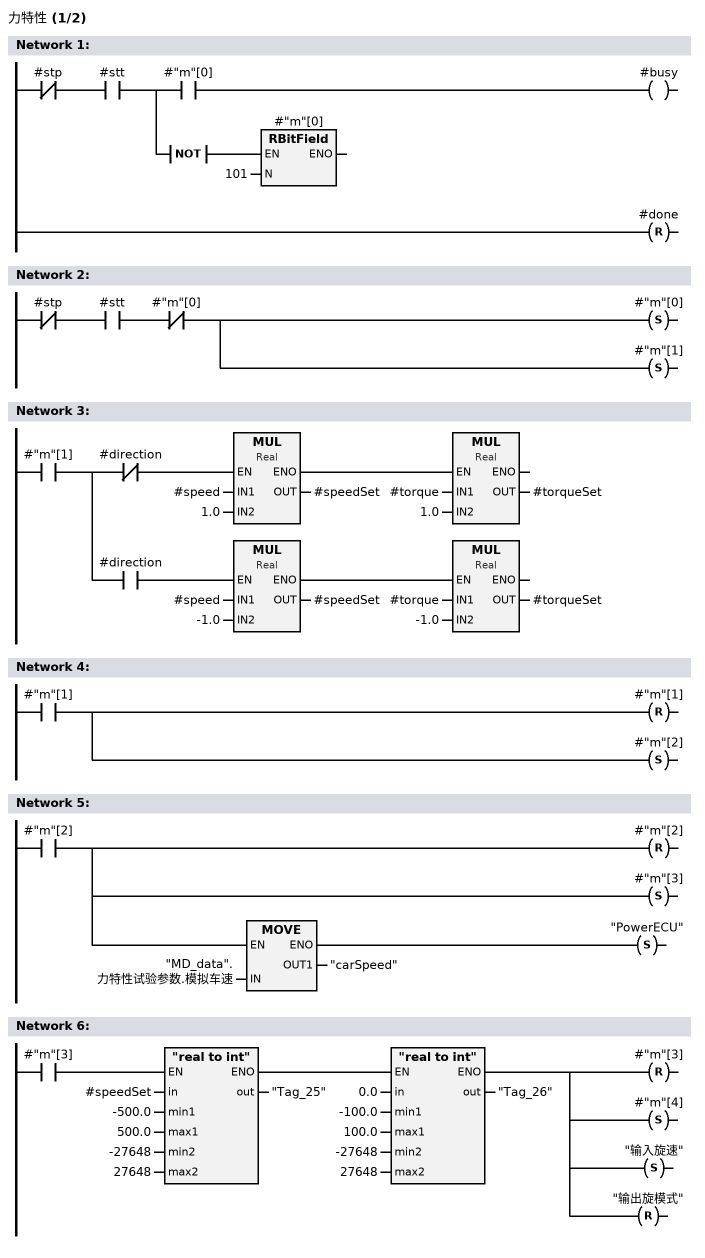
   // no SCL statement known for RBitField: written as a call
   #_w1 := NOT #stp AND #stt;
   #busy := #_w1 AND #"m"[0];
   IF NOT #_w1 THEN RBitField(n := 101, operand := #"m"[0]); END_IF;
   #done := FALSE;
END_REGION

REGION Network 2
   RUNG wire#powerrail
      I_Contact( #stp )
      Contact( #stt )
      I_Contact( #"m"[0] )
      wire#w1
      S_Coil( #"m"[0] )
   END_RUNG
   RUNG wire#w1
      S_Coil( #"m"[1] )
   END_RUNG
   // the same network as SCL:
   #_w1 := NOT #stp AND #stt AND NOT #"m"[0];
   IF #_w1 THEN
       #"m"[0] := TRUE;
       #"m"[1] := TRUE;
   END_IF;
END_REGION

REGION Network 3
   RUNG wire#powerrail
      Contact( #"m"[1] )
      wire#w1
      I_Contact( #direction )
      { S7_Templates := "SrcType := Real" } Mul(in1 := #speed, in2 := 1.0, out => #speedSet)
      { S7_Templates := "SrcType := Real" } Mul(in1 := #torque, in2 := 1.0, out => #torqueSet)
   END_RUNG
   RUNG wire#w1
      Contact( #direction )
      { S7_Templates := "SrcType := Real" } Mul(in1 := #speed, in2 := -1.0, out => #speedSet)
      { S7_Templates := "SrcType := Real" } Mul(in1 := #torque, in2 := -1.0, out => #torqueSet)
   END_RUNG
   // the same network as SCL:
   IF #"m"[1] AND NOT #direction THEN
       #speedSet := #speed * 1.0;
       #torqueSet := #torque * 1.0;
   END_IF;
   IF #"m"[1] AND #direction THEN
       #speedSet := #speed * (-1.0);
       #torqueSet := #torque * (-1.0);
   END_IF;
END_REGION

REGION Network 4
   RUNG wire#powerrail
      Contact( #"m"[1] )
      wire#w1
      R_Coil( #"m"[1] )
   END_RUNG
   RUNG wire#w1
      S_Coil( #"m"[2] )
   END_RUNG
   // the same network as SCL:
   #_w1 := #"m"[1];
   IF #_w1 THEN
       #"m"[1] := FALSE;
       #"m"[2] := TRUE;
   END_IF;
END_REGION

REGION Network 5
   RUNG wire#powerrail
      Contact( #"m"[2] )
      wire#w1
      R_Coil( #"m"[2] )
   END_RUNG
   RUNG wire#w1
      S_Coil( #"m"[3] )
   END_RUNG
   RUNG wire#w1
      Move(in := "MD_data".力特性试验参数.模拟车速, out1 => "carSpeed")
      S_Coil( "PowerECU" )
   END_RUNG
   // the same network as SCL:
   #_w1 := #"m"[2];
   IF #_w1 THEN
       #"m"[2] := FALSE;
       #"m"[3] := TRUE;
       "carSpeed" := "MD_data".力特性试验参数.模拟车速;
       "PowerECU" := TRUE;
   END_IF;
END_REGION

REGION Network 6
   RUNG wire#powerrail
      Contact( #"m"[3] )
      "real to int"(in := #speedSet, min1 := -500.0, max1 := 500.0, min2 := -27648, max2 := 27648, out => "Tag_25")
      "real to int"(in := 0.0, min1 := -100.0, max1 := 100.0, min2 := -27648, max2 := 27648, out => "Tag_26")
      wire#w1
      R_Coil( #"m"[3] )
   END_RUNG
   RUNG wire#w1
      S_Coil( #"m"[4] )
   END_RUNG
   RUNG wire#w1
      S_Coil( "输入旋速" )
   END_RUNG
   RUNG wire#w1
      R_Coil( "输出旋模式" )
   END_RUNG
   // the same network as SCL:
   "real to int"(EN := #"m"[3],
                 in := #speedSet,
                 min1 := -500.0,
                 max1 := 500.0,
                 min2 := -27648,
                 max2 := 27648,
                 out => "Tag_25",
                 ENO => #_w1);
   "real to int"(EN := #_w1,
                 in := 0.0,
                 min1 := -100.0,
                 max1 := 100.0,
                 min2 := -27648,
                 max2 := 27648,
                 out => "Tag_26",
                 ENO => #_w2);
   IF #_w2 THEN
       #"m"[3] := FALSE;
       #"m"[4] := TRUE;
       "输入旋速" := TRUE;
       "输出旋模式" := FALSE;
   END_IF;
END_REGION

REGION Network 7
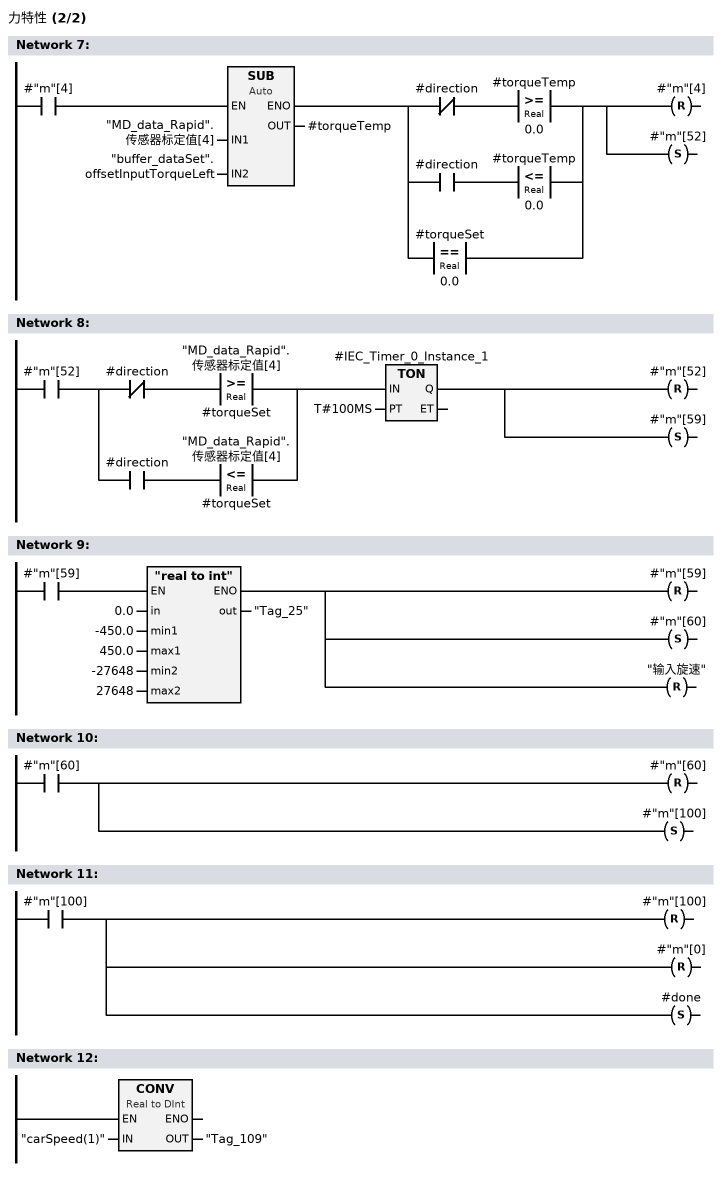
   RUNG wire#powerrail
      Contact( #"m"[4] )
      Sub(in1 := "MD_data_Rapid".传感器标定值[4], in2 := "buffer_dataSet".offsetInputTorqueLeft, out => #torqueTemp)
      wire#w1
      I_Contact( #direction )
      { S7_Templates := "SrcType := Real" } GE_Contact(in1 := #torqueTemp, in2 := 0.0)
      wire#w2
      R_Coil( #"m"[4] )
   END_RUNG
   RUNG wire#w1
      Contact( #direction )
      { S7_Templates := "SrcType := Real" } LE_Contact(in1 := #torqueTemp, in2 := 0.0)
   END_RUNG wire#w2
   RUNG wire#w1
      { S7_Templates := "SrcType := Real" } EQ_Contact(in1 := #torqueSet, in2 := 0.0)
   END_RUNG wire#w2
   RUNG wire#w2
      S_Coil( #"m"[52] )
   END_RUNG
   // the same network as SCL:
   IF #"m"[4] THEN #torqueTemp := "MD_data_Rapid".传感器标定值[4] - "buffer_dataSet".offsetInputTorqueLeft; END_IF;
   #_w1 := #"m"[4] AND ((NOT #direction AND (#torqueTemp >= 0.0)) OR (#direction AND (#torqueTemp <= 0.0)) OR (#torqueSet = 0.0));
   IF #_w1 THEN
       #"m"[4] := FALSE;
       #"m"[52] := TRUE;
   END_IF;
END_REGION

REGION Network 8
   #IEC_Timer_0_Instance_1(IN := #"m"[52] AND ((NOT #direction AND ("MD_data_Rapid".传感器标定值[4] >= #torqueSet)) OR (#direction AND ("MD_data_Rapid".传感器标定值[4] <= #torqueSet))),   // TON
                           PT := T#100MS);
   IF #IEC_Timer_0_Instance_1.Q THEN
       #"m"[52] := FALSE;
       #"m"[59] := TRUE;
   END_IF;
END_REGION

REGION Network 9
   RUNG wire#powerrail
      Contact( #"m"[59] )
      "real to int"(in := 0.0, min1 := -450.0, max1 := 450.0, min2 := -27648, max2 := 27648, out => "Tag_25")
      wire#w1
      R_Coil( #"m"[59] )
   END_RUNG
   RUNG wire#w1
      S_Coil( #"m"[60] )
   END_RUNG
   RUNG wire#w1
      R_Coil( "输入旋速" )
   END_RUNG
   // the same network as SCL:
   "real to int"(EN := #"m"[59],
                 in := 0.0,
                 min1 := -450.0,
                 max1 := 450.0,
                 min2 := -27648,
                 max2 := 27648,
                 out => "Tag_25",
                 ENO => #_w1);
   IF #_w1 THEN
       #"m"[59] := FALSE;
       #"m"[60] := TRUE;
       "输入旋速" := FALSE;
   END_IF;
END_REGION

REGION Network 10
   RUNG wire#powerrail
      Contact( #"m"[60] )
      wire#w1
      R_Coil( #"m"[60] )
   END_RUNG
   RUNG wire#w1
      S_Coil( #"m"[100] )
   END_RUNG
   // the same network as SCL:
   #_w1 := #"m"[60];
   IF #_w1 THEN
       #"m"[60] := FALSE;
       #"m"[100] := TRUE;
   END_IF;
END_REGION

REGION Network 11
   RUNG wire#powerrail
      Contact( #"m"[100] )
      wire#w1
      R_Coil( #"m"[100] )
   END_RUNG
   RUNG wire#w1
      R_Coil( #"m"[0] )
   END_RUNG
   RUNG wire#w1
      S_Coil( #done )
   END_RUNG
   // the same network as SCL:
   #_w1 := #"m"[100];
   IF #_w1 THEN
       #"m"[100] := FALSE;
       #"m"[0] := FALSE;
       #done := TRUE;
   END_IF;
END_REGION

REGION Network 12
   RUNG wire#powerrail
      { S7_Templates := "[SrcType := Real, DestType := DInt]" } Convert(in := "carSpeed(1)", out => "Tag_109")
   END_RUNG
   // the same network as SCL:
   "Tag_109" := REAL_TO_DINT("carSpeed(1)");
END_REGION
END_FUNCTION_BLOCK

FUNCTION_BLOCK "逆向空载"   // FB10, LAD
{ S7_Optimized_Access := 'TRUE' }
VERSION : 0.1
   VAR_INPUT
      stt : Bool;
      stp : Bool;
      direction : Bool;
      speed : Real;
      angle : Real;
   END_VAR
   VAR_OUTPUT
      done : Bool;
      error : Bool;
      busy : Bool;
   END_VAR
   VAR
      "m" : Array[0..100] of Bool;
      "time" : IEC_TIMER;
      newCV : DInt;
      angleSet : Real;
      speedSet : Real;
      angleRead : Real;
   END_VAR
   VAR_TEMP   // added for the SCL form of the ladder/FBD networks
      _w1 : Bool;
      _w2 : Bool;
   END_VAR
BEGIN

REGION Network 1
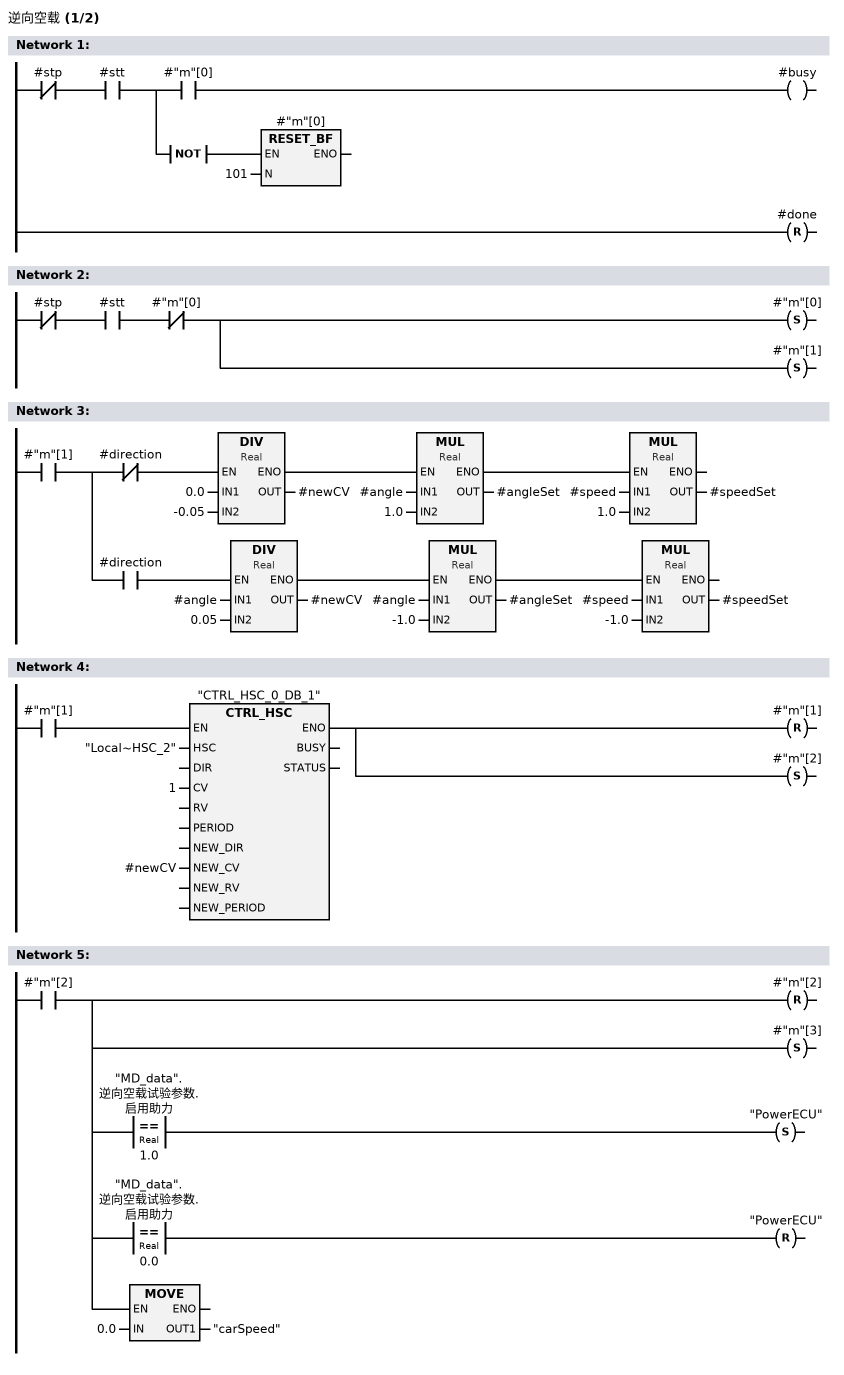
   // no SCL statement known for RBitfield: written as a call
   #_w1 := NOT #stp AND #stt;
   #busy := #_w1 AND #"m"[0];
   IF NOT #_w1 THEN RESET_BF(operand := #"m"[0], n := 101); END_IF;
   #done := FALSE;
END_REGION

REGION Network 2
   RUNG wire#powerrail
      I_Contact( #stp )
      Contact( #stt )
      I_Contact( #"m"[0] )
      wire#w1
      S_Coil( #"m"[0] )
   END_RUNG
   RUNG wire#w1
      S_Coil( #"m"[1] )
   END_RUNG
   // the same network as SCL:
   #_w1 := NOT #stp AND #stt AND NOT #"m"[0];
   IF #_w1 THEN
       #"m"[0] := TRUE;
       #"m"[1] := TRUE;
   END_IF;
END_REGION

REGION Network 3
   RUNG wire#powerrail
      Contact( #"m"[1] )
      wire#w1
      I_Contact( #direction )
      { S7_Templates := "SrcType := Real" } Div(in1 := 0.0, in2 := -0.05, out => #newCV)
      { S7_Templates := "SrcType := Real" } Mul(in1 := #angle, in2 := 1.0, out => #angleSet)
      { S7_Templates := "SrcType := Real" } Mul(in1 := #speed, in2 := 1.0, out => #speedSet)
   END_RUNG
   RUNG wire#w1
      Contact( #direction )
      { S7_Templates := "SrcType := Real" } Div(in1 := #angle, in2 := 0.05, out => #newCV)
      { S7_Templates := "SrcType := Real" } Mul(in1 := #angle, in2 := -1.0, out => #angleSet)
      { S7_Templates := "SrcType := Real" } Mul(in1 := #speed, in2 := -1.0, out => #speedSet)
   END_RUNG
   // the same network as SCL:
   IF #"m"[1] AND NOT #direction THEN
       #newCV := 0.0 / (-0.05);
       #angleSet := #angle * 1.0;
       #speedSet := #speed * 1.0;
   END_IF;
   IF #"m"[1] AND #direction THEN
       #newCV := #angle / 0.05;
       #angleSet := #angle * (-1.0);
       #speedSet := #speed * (-1.0);
   END_IF;
END_REGION

REGION Network 4
   // ENO of a box is taken as its EN; it also drops when the box reports an error
   IF #"m"[1] THEN
       "CTRL_HSC_0_DB_1"(HSC := "Local~HSC_2", CV := 1, NEW_CV := #newCV);   // CTRL_HSC
   END_IF;
   #_w1 := #"m"[1];
   IF #_w1 THEN
       #"m"[1] := FALSE;
       #"m"[2] := TRUE;
   END_IF;
END_REGION

REGION Network 5
   RUNG wire#powerrail
      Contact( #"m"[2] )
      wire#w1
      R_Coil( #"m"[2] )
   END_RUNG
   RUNG wire#w1
      S_Coil( #"m"[3] )
   END_RUNG
   RUNG wire#w1
      { S7_Templates := "SrcType := Real" } EQ_Contact(in1 := "MD_data".逆向空载试验参数.启用助力, in2 := 1.0)
      S_Coil( "PowerECU" )
   END_RUNG
   RUNG wire#w1
      { S7_Templates := "SrcType := Real" } EQ_Contact(in1 := "MD_data".逆向空载试验参数.启用助力, in2 := 0.0)
      R_Coil( "PowerECU" )
   END_RUNG
   RUNG wire#w1
      Move(in := 0.0, out1 => "carSpeed")
   END_RUNG
   // the same network as SCL:
   #_w1 := #"m"[2];
   IF #_w1 THEN
       #"m"[2] := FALSE;
       #"m"[3] := TRUE;
   END_IF;
   IF #_w1 AND ("MD_data".逆向空载试验参数.启用助力 = 1.0) THEN "PowerECU" := TRUE; END_IF;
   IF #_w1 AND ("MD_data".逆向空载试验参数.启用助力 = 0.0) THEN "PowerECU" := FALSE; END_IF;
   IF #_w1 THEN "carSpeed" := 0.0; END_IF;
END_REGION

REGION Network 7
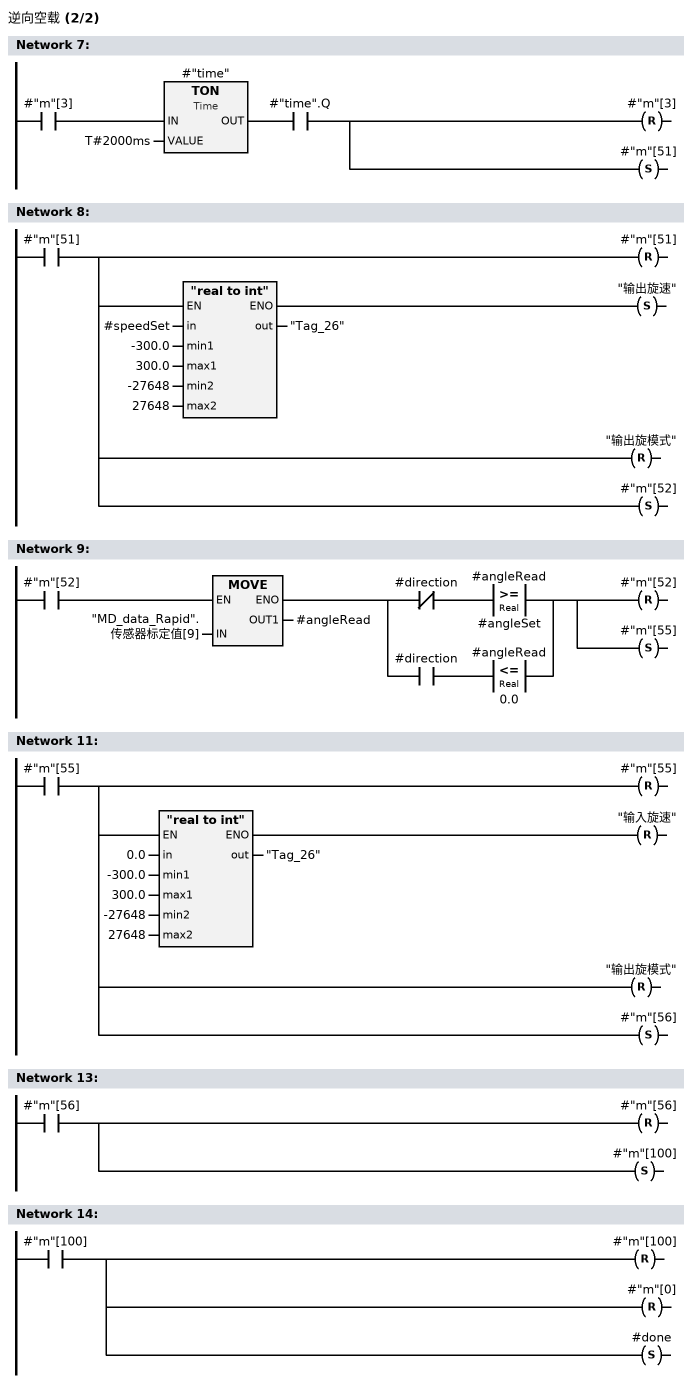
   #"time".TON(IN := #"m"[3], PT := T#2000ms);   // TON coil
   #_w1 := #"m"[3] AND #"time".Q;
   IF #_w1 THEN
       #"m"[3] := FALSE;
       #"m"[51] := TRUE;
   END_IF;
END_REGION

REGION Network 8
   RUNG wire#powerrail
      Contact( #"m"[51] )
      wire#w1
      R_Coil( #"m"[51] )
   END_RUNG
   RUNG wire#w1
      "real to int"(in := #speedSet, min1 := -300.0, max1 := 300.0, min2 := -27648, max2 := 27648, out => "Tag_26")
      S_Coil( "输出旋速" )
   END_RUNG
   RUNG wire#w1
      R_Coil( "输出旋模式" )
   END_RUNG
   RUNG wire#w1
      S_Coil( #"m"[52] )
   END_RUNG
   // the same network as SCL:
   #_w1 := #"m"[51];
   IF #_w1 THEN #"m"[51] := FALSE; END_IF;
   "real to int"(EN := #_w1,
                 in := #speedSet,
                 min1 := -300.0,
                 max1 := 300.0,
                 min2 := -27648,
                 max2 := 27648,
                 out => "Tag_26",
                 ENO => #_w2);
   IF #_w2 THEN "输出旋速" := TRUE; END_IF;
   IF #_w1 THEN
       "输出旋模式" := FALSE;
       #"m"[52] := TRUE;
   END_IF;
END_REGION

REGION Network 9
   RUNG wire#powerrail
      Contact( #"m"[52] )
      Move(in := "MD_data_Rapid".传感器标定值[9], out1 => #angleRead)
      wire#w1
      I_Contact( #direction )
      { S7_Templates := "SrcType := Real" } GE_Contact(in1 := #angleRead, in2 := #angleSet)
      wire#w2
      R_Coil( #"m"[52] )
   END_RUNG
   RUNG wire#w1
      Contact( #direction )
      { S7_Templates := "SrcType := Real" } LE_Contact(in1 := #angleRead, in2 := 0.0)
   END_RUNG wire#w2
   RUNG wire#w2
      S_Coil( #"m"[55] )
   END_RUNG
   // the same network as SCL:
   IF #"m"[52] THEN #angleRead := "MD_data_Rapid".传感器标定值[9]; END_IF;
   #_w1 := #"m"[52] AND ((NOT #direction AND (#angleRead >= #angleSet)) OR (#direction AND (#angleRead <= 0.0)));
   IF #_w1 THEN
       #"m"[52] := FALSE;
       #"m"[55] := TRUE;
   END_IF;
END_REGION

REGION Network 11
   RUNG wire#powerrail
      Contact( #"m"[55] )
      wire#w1
      R_Coil( #"m"[55] )
   END_RUNG
   RUNG wire#w1
      "real to int"(in := 0.0, min1 := -300.0, max1 := 300.0, min2 := -27648, max2 := 27648, out => "Tag_26")
      R_Coil( "输入旋速" )
   END_RUNG
   RUNG wire#w1
      R_Coil( "输出旋模式" )
   END_RUNG
   RUNG wire#w1
      S_Coil( #"m"[56] )
   END_RUNG
   // the same network as SCL:
   #_w1 := #"m"[55];
   IF #_w1 THEN #"m"[55] := FALSE; END_IF;
   "real to int"(EN := #_w1,
                 in := 0.0,
                 min1 := -300.0,
                 max1 := 300.0,
                 min2 := -27648,
                 max2 := 27648,
                 out => "Tag_26",
                 ENO => #_w2);
   IF #_w2 THEN "输入旋速" := FALSE; END_IF;
   IF #_w1 THEN
       "输出旋模式" := FALSE;
       #"m"[56] := TRUE;
   END_IF;
END_REGION

REGION Network 13
   RUNG wire#powerrail
      Contact( #"m"[56] )
      wire#w1
      R_Coil( #"m"[56] )
   END_RUNG
   RUNG wire#w1
      S_Coil( #"m"[100] )
   END_RUNG
   // the same network as SCL:
   #_w1 := #"m"[56];
   IF #_w1 THEN
       #"m"[56] := FALSE;
       #"m"[100] := TRUE;
   END_IF;
END_REGION

REGION Network 14
   RUNG wire#powerrail
      Contact( #"m"[100] )
      wire#w1
      R_Coil( #"m"[100] )
   END_RUNG
   RUNG wire#w1
      R_Coil( #"m"[0] )
   END_RUNG
   RUNG wire#w1
      S_Coil( #done )
   END_RUNG
   // the same network as SCL:
   #_w1 := #"m"[100];
   IF #_w1 THEN
       #"m"[100] := FALSE;
       #"m"[0] := FALSE;
       #done := TRUE;
   END_IF;
END_REGION
END_FUNCTION_BLOCK

FUNCTION_BLOCK "固定工件"   // FB11, LAD
{ S7_Optimized_Access := 'TRUE' }
VERSION : 0.1
   VAR_INPUT
      stt : Bool;
      stp : Bool;
   END_VAR
   VAR_OUTPUT
      done : Bool;
      error : Bool;
      busy : Bool;
   END_VAR
   VAR
      "m" : Array[0..100] of Bool;
      "time" : Real;
      partCount : Real;
      speedSet : Real;
      timeSet : Real;
      loadSet : Real;
      carSpeed : Real;
      IEC_Timer_0_Instance : TON_TIME;
   END_VAR
   VAR_TEMP   // added for the SCL form of the ladder/FBD networks
      _w1 : Bool;
   END_VAR
BEGIN

REGION Network 1
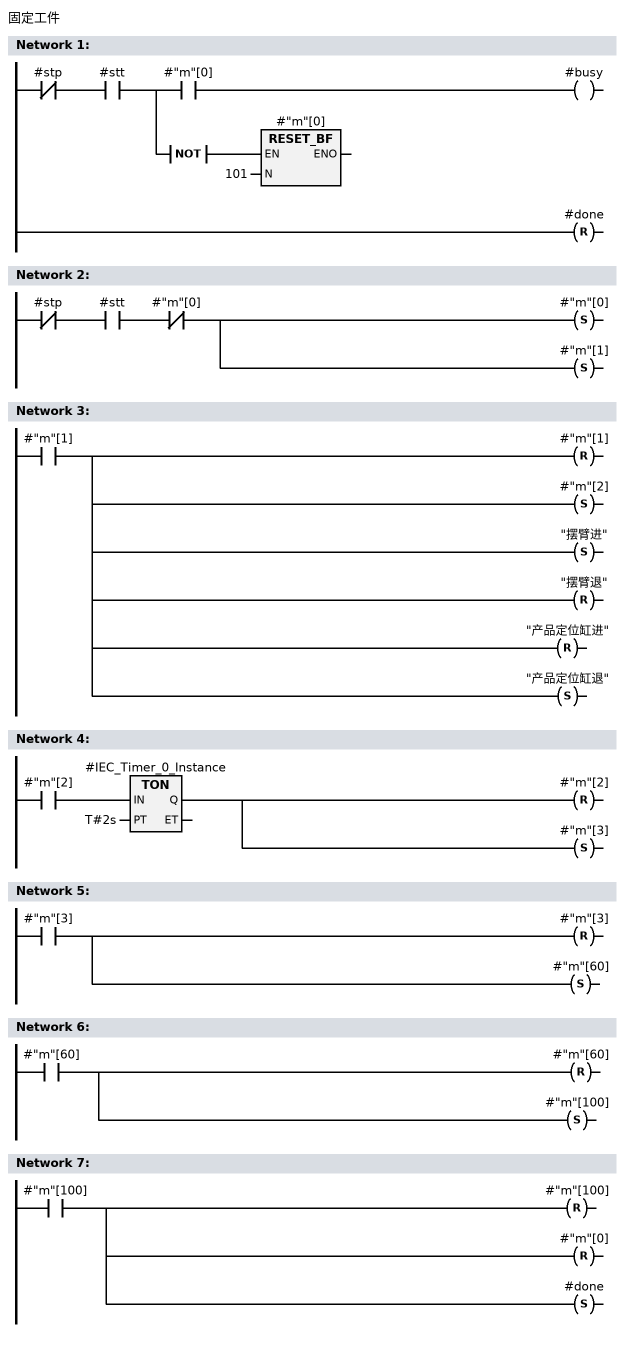
   // no SCL statement known for RBitfield: written as a call
   #_w1 := NOT #stp AND #stt;
   #busy := #_w1 AND #"m"[0];
   IF NOT #_w1 THEN RESET_BF(operand := #"m"[0], n := 101); END_IF;
   #done := FALSE;
END_REGION

REGION Network 2
   RUNG wire#powerrail
      I_Contact( #stp )
      Contact( #stt )
      I_Contact( #"m"[0] )
      wire#w1
      S_Coil( #"m"[0] )
   END_RUNG
   RUNG wire#w1
      S_Coil( #"m"[1] )
   END_RUNG
   // the same network as SCL:
   #_w1 := NOT #stp AND #stt AND NOT #"m"[0];
   IF #_w1 THEN
       #"m"[0] := TRUE;
       #"m"[1] := TRUE;
   END_IF;
END_REGION

REGION Network 3
   RUNG wire#powerrail
      Contact( #"m"[1] )
      wire#w1
      R_Coil( #"m"[1] )
   END_RUNG
   RUNG wire#w1
      S_Coil( #"m"[2] )
   END_RUNG
   RUNG wire#w1
      S_Coil( "摆臂进" )
   END_RUNG
   RUNG wire#w1
      R_Coil( "摆臂退" )
   END_RUNG
   RUNG wire#w1
      R_Coil( "产品定位缸进" )
   END_RUNG
   RUNG wire#w1
      S_Coil( "产品定位缸退" )
   END_RUNG
   // the same network as SCL:
   #_w1 := #"m"[1];
   IF #_w1 THEN
       #"m"[1] := FALSE;
       #"m"[2] := TRUE;
       "摆臂进" := TRUE;
       "摆臂退" := FALSE;
       "产品定位缸进" := FALSE;
       "产品定位缸退" := TRUE;
   END_IF;
END_REGION

REGION Network 4
   #IEC_Timer_0_Instance(IN := #"m"[2], PT := T#2s);   // TON
   IF #IEC_Timer_0_Instance.Q THEN
       #"m"[2] := FALSE;
       #"m"[3] := TRUE;
   END_IF;
END_REGION

REGION Network 5
   RUNG wire#powerrail
      Contact( #"m"[3] )
      wire#w1
      R_Coil( #"m"[3] )
   END_RUNG
   RUNG wire#w1
      S_Coil( #"m"[60] )
   END_RUNG
   // the same network as SCL:
   #_w1 := #"m"[3];
   IF #_w1 THEN
       #"m"[3] := FALSE;
       #"m"[60] := TRUE;
   END_IF;
END_REGION

REGION Network 6
   RUNG wire#powerrail
      Contact( #"m"[60] )
      wire#w1
      R_Coil( #"m"[60] )
   END_RUNG
   RUNG wire#w1
      S_Coil( #"m"[100] )
   END_RUNG
   // the same network as SCL:
   #_w1 := #"m"[60];
   IF #_w1 THEN
       #"m"[60] := FALSE;
       #"m"[100] := TRUE;
   END_IF;
END_REGION

REGION Network 7
   RUNG wire#powerrail
      Contact( #"m"[100] )
      wire#w1
      R_Coil( #"m"[100] )
   END_RUNG
   RUNG wire#w1
      R_Coil( #"m"[0] )
   END_RUNG
   RUNG wire#w1
      S_Coil( #done )
   END_RUNG
   // the same network as SCL:
   #_w1 := #"m"[100];
   IF #_w1 THEN
       #"m"[100] := FALSE;
       #"m"[0] := FALSE;
       #done := TRUE;
   END_IF;
END_REGION
END_FUNCTION_BLOCK

FUNCTION_BLOCK "振动检测"   // FB12, LAD
{ S7_Optimized_Access := 'TRUE' }
VERSION : 0.1
   VAR_INPUT
      stt : Bool;
      stp : Bool;
   END_VAR
   VAR_OUTPUT
      done : Bool;
      error : Bool;
      busy : Bool;
   END_VAR
   VAR
      "m" : Array[0..100] of Bool;
      "time" : IEC_TIMER;
      time_1 : IEC_TIMER;
      speedC : Real;
      IEC_Timer_0_Instance : TON_TIME;
      IEC_Timer_0_Instance_1 : TON_TIME;
      IEC_Timer_0_Instance_2 : TON_TIME;
      IEC_Timer_0_Instance_3 : TON_TIME;
      IEC_Timer_0_Instance_4 : TON_TIME;
      IEC_Timer_0_Instance_5 : TON_TIME;
   END_VAR
   VAR_TEMP
      done1 : Bool;
      done2 : Bool;
      done3 : Bool;
      done4 : Bool;
      n : Bool;
      n_1 : Bool;
      lang : Real;
   END_VAR
   VAR_TEMP   // added for the SCL form of the ladder/FBD networks
      _w1 : Bool;
      _w2 : Bool;
      _w3 : Bool;
   END_VAR
BEGIN

REGION Network 1
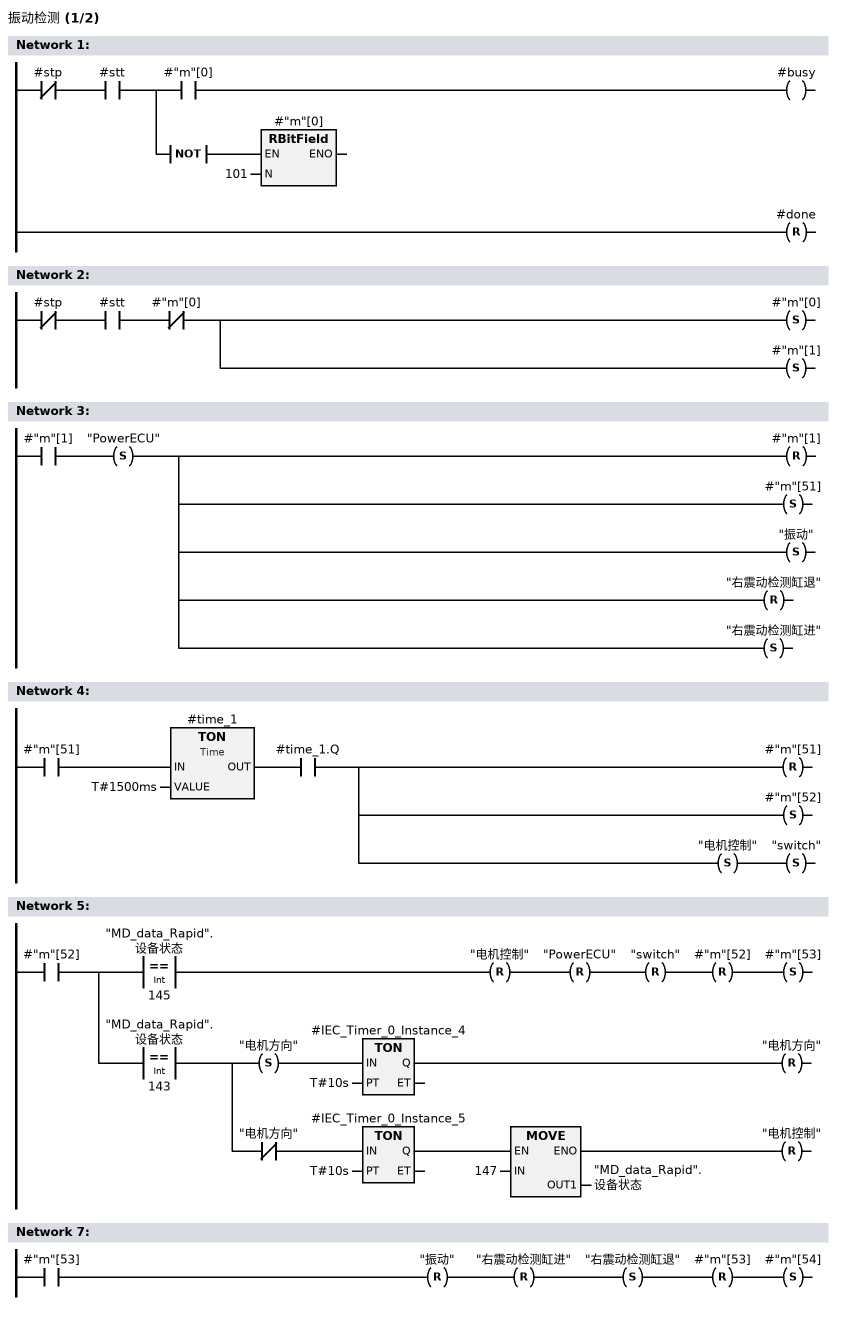
   // no SCL statement known for RBitField: written as a call
   #_w1 := NOT #stp AND #stt;
   #busy := #_w1 AND #"m"[0];
   IF NOT #_w1 THEN RBitField(n := 101, operand := #"m"[0]); END_IF;
   #done := FALSE;
END_REGION

REGION Network 2
   RUNG wire#powerrail
      I_Contact( #stp )
      Contact( #stt )
      I_Contact( #"m"[0] )
      wire#w1
      S_Coil( #"m"[0] )
   END_RUNG
   RUNG wire#w1
      S_Coil( #"m"[1] )
   END_RUNG
   // the same network as SCL:
   #_w1 := NOT #stp AND #stt AND NOT #"m"[0];
   IF #_w1 THEN
       #"m"[0] := TRUE;
       #"m"[1] := TRUE;
   END_IF;
END_REGION

REGION Network 3
   RUNG wire#powerrail
      Contact( #"m"[1] )
      S_Coil( "PowerECU" )
      wire#w1
      R_Coil( #"m"[1] )
   END_RUNG
   RUNG wire#w1
      S_Coil( #"m"[51] )
   END_RUNG
   RUNG wire#w1
      S_Coil( "振动" )
   END_RUNG
   RUNG wire#w1
      R_Coil( "右震动检测缸退" )
   END_RUNG
   RUNG wire#w1
      S_Coil( "右震动检测缸进" )
   END_RUNG
   // the same network as SCL:
   IF #"m"[1] THEN "PowerECU" := TRUE; END_IF;
   #_w1 := #"m"[1];
   IF #_w1 THEN
       #"m"[1] := FALSE;
       #"m"[51] := TRUE;
       "振动" := TRUE;
       "右震动检测缸退" := FALSE;
       "右震动检测缸进" := TRUE;
   END_IF;
END_REGION

REGION Network 4
   #time_1.TON(IN := #"m"[51], PT := T#1500ms);   // TON coil
   #_w1 := #"m"[51] AND #time_1.Q;
   IF #_w1 THEN
       #"m"[51] := FALSE;
       #"m"[52] := TRUE;
       "电机控制" := TRUE;
       "switch" := TRUE;
   END_IF;
END_REGION

REGION Network 5
   IF #"m"[52] AND ("MD_data_Rapid".设备状态 = 145) THEN
       "电机控制" := FALSE;
       "PowerECU" := FALSE;
       "switch" := FALSE;
   END_IF;
   #_w1 := #"m"[52] AND ("MD_data_Rapid".设备状态 = 145);
   #_w2 := #"m"[52];
   IF #_w1 THEN
       #"m"[52] := FALSE;
       #"m"[53] := TRUE;
   END_IF;
   #_w3 := #_w2 AND ("MD_data_Rapid".设备状态 = 143);
   IF #_w3 THEN "电机方向" := TRUE; END_IF;
   #IEC_Timer_0_Instance_4(IN := #_w3, PT := T#10s);   // TON
   IF #IEC_Timer_0_Instance_4.Q THEN "电机方向" := FALSE; END_IF;
   #IEC_Timer_0_Instance_5(IN := #_w3 AND NOT "电机方向", PT := T#10s);   // TON
   IF #IEC_Timer_0_Instance_5.Q THEN
       "MD_data_Rapid".设备状态 := 147;
       "电机控制" := FALSE;
   END_IF;
END_REGION

REGION Network 7
   RUNG wire#powerrail
      Contact( #"m"[53] )
      R_Coil( "振动" )
      R_Coil( "右震动检测缸进" )
      S_Coil( "右震动检测缸退" )
      R_Coil( #"m"[53] )
      S_Coil( #"m"[54] )
   END_RUNG
   // the same network as SCL:
   IF #"m"[53] THEN
       "振动" := FALSE;
       "右震动检测缸进" := FALSE;
       "右震动检测缸退" := TRUE;
   END_IF;
   #_w1 := #"m"[53];
   IF #_w1 THEN
       #"m"[53] := FALSE;
       #"m"[54] := TRUE;
   END_IF;
END_REGION

REGION Network 8
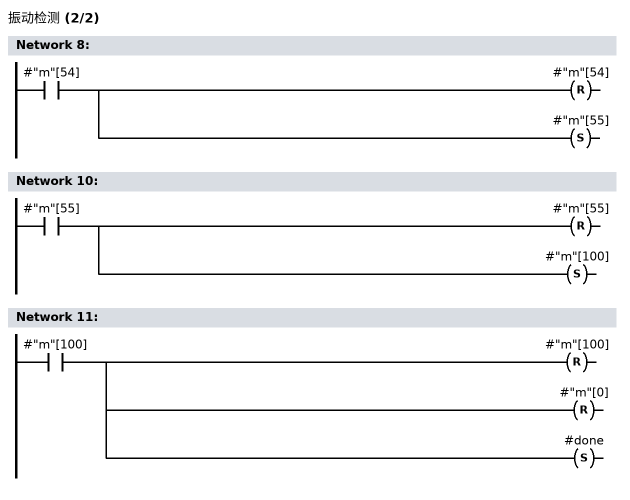
   RUNG wire#powerrail
      Contact( #"m"[54] )
      wire#w1
      R_Coil( #"m"[54] )
   END_RUNG
   RUNG wire#w1
      S_Coil( #"m"[55] )
   END_RUNG
   // the same network as SCL:
   #_w1 := #"m"[54];
   IF #_w1 THEN
       #"m"[54] := FALSE;
       #"m"[55] := TRUE;
   END_IF;
END_REGION

REGION Network 10
   RUNG wire#powerrail
      Contact( #"m"[55] )
      wire#w1
      R_Coil( #"m"[55] )
   END_RUNG
   RUNG wire#w1
      S_Coil( #"m"[100] )
   END_RUNG
   // the same network as SCL:
   #_w1 := #"m"[55];
   IF #_w1 THEN
       #"m"[55] := FALSE;
       #"m"[100] := TRUE;
   END_IF;
END_REGION

REGION Network 11
   RUNG wire#powerrail
      Contact( #"m"[100] )
      wire#w1
      R_Coil( #"m"[100] )
   END_RUNG
   RUNG wire#w1
      R_Coil( #"m"[0] )
   END_RUNG
   RUNG wire#w1
      S_Coil( #done )
   END_RUNG
   // the same network as SCL:
   #_w1 := #"m"[100];
   IF #_w1 THEN
       #"m"[100] := FALSE;
       #"m"[0] := FALSE;
       #done := TRUE;
   END_IF;
END_REGION
END_FUNCTION_BLOCK

FUNCTION_BLOCK "auto_100"   // FB13, LAD
{ S7_Optimized_Access := 'TRUE' }
VERSION : 0.1
   VAR_INPUT
      stt : Bool;
      stp : Bool;
   END_VAR
   VAR_OUTPUT
      done : Bool;
      error : Bool;
      busy : Bool;
   END_VAR
   VAR
      "m" : Array[0..100] of Bool;
      "time" : IEC_TIMER;
      time_1 : IEC_TIMER;
   END_VAR
   VAR_TEMP
      done1 : Bool;
      done2 : Bool;
      done3 : Bool;
      done4 : Bool;
      n : Bool;
      n_1 : Bool;
   END_VAR
   VAR_TEMP   // added for the SCL form of the ladder/FBD networks
      _w1 : Bool;
   END_VAR
BEGIN

REGION Network 1
